LIN {X 0,Y 287.077,Z 619.166,A -85,B 0,C 180,E1 -18390.734,E2 -18390.734} C_VEL
LIN {X 0,Y 290.239,Z 606.893,A -85,B 0,C 180,E1 -18391.78,E2 -18391.78} C_VEL
LIN {X 0,Y 292.756,Z 594.998,A -85,B 0,C 180,E1 -18392.54,E2 -18392.54} C_VEL
LIN {X 0,Y 304.333,Z 525.318,A -85,B 0,C 180,E1 -18395.699,E2 -18395.699} C_VEL
LIN {X 0,Y 304.333,Z 521.564,A -85,B 0,C 180,E1 -18396.179,E2 -18396.179} C_VEL
LIN {X 0,Y 302.945,Z 516.848,A -85,B 0,C 180,E1 -18397.582,E2 -18397.582} C_VEL
LIN {X 0,Y 301.83,Z 513.451,A -85,B 0,C 180,E1 -18398.873,E2 -18398.873} C_VEL
LIN {X 0,Y 300.898,Z 510.648,A -85,B 0,C 180,E1 -18400.235,E2 -18400.235} C_VEL
LIN {X 0,Y 299.797,Z 507.286,A -85,B 0,C 180,E1 -18402.831,E2 -18402.831} C_VEL
LIN {X 0,Y 299.555,Z 506.287,A -85,B 0,C 180,E1 -18404.736,E2 -18404.736} C_VEL
LIN {X 0,Y 300.178,Z 506.371,A -85,B 0,C 180,E1 -18407.424,E2 -18407.424} C_VEL
LIN {X 0,Y 301.713,Z 507.829,A -85,B 0,C 180,E1 -18409.732,E2 -18409.732} C_VEL
LIN {X 0,Y 303.161,Z 509.629,A -85,B 0,C 180,E1 -18411.25,E2 -18411.25} C_VEL
LIN {X 0,Y 303.675,Z 510.855,A -85,B 0,C 180,E1 -18411.798,E2 -18411.798} C_VEL
LIN {X 0,Y 303.632,Z 512.913,A -85,B 0,C 180,E1 -18412.113,E2 -18412.113} C_VEL
LIN {X 0,Y 302.89,Z 524.787,A -85,B 0,C 180,E1 -18413.442,E2 -18413.442} C_VEL
LIN {X 0,Y 301.946,Z 536.286,A -85,B 0,C 180,E1 -18414.495,E2 -18414.495} C_VEL
LIN {X 0,Y 300.792,Z 545.281,A -85,B 0,C 180,E1 -18415.064,E2 -18415.064} C_VEL
LIN {X 0,Y 290.965,Z 604.012,A -85,B 0,C 180,E1 -18417.747,E2 -18417.747} C_VEL
LIN {X 0,Y 287.846,Z 617.704,A -85,B 0,C 180,E1 -18418.592,E2 -18418.592} C_VEL
LIN {X 0,Y 284.125,Z 631.372,A -85,B 0,C 180,E1 -18419.736,E2 -18419.736} C_VEL
LIN {X 0,Y 280.163,Z 643.742,A -85,B 0,C 180,E1 -18421.125,E2 -18421.125} C_VEL
LIN {X 0,Y 276.068,Z 655.019,A -85,B 0,C 180,E1 -18422.727,E2 -18422.727} C_VEL
LIN {X 0,Y 272.401,Z 664.289,A -85,B 0,C 180,E1 -18424.396,E2 -18424.396} C_VEL
LIN {X 0,Y 268.548,Z 673.397,A -85,B 0,C 180,E1 -18426.436,E2 -18426.436} C_VEL
LIN {X 0,Y 265.028,Z 681.094,A -85,B 0,C 180,E1 -18428.616,E2 -18428.616} C_VEL
LIN {X 0,Y 261.491,Z 688.208,A -85,B 0,C 180,E1 -18431.185,E2 -18431.185} C_VEL
LIN {X 0,Y 259.222,Z 692.983,A -85,B 0,C 180,E1 -18433.46,E2 -18433.46} C_VEL
LIN {X 0,Y 257.36,Z 696.664,A -85,B 0,C 180,E1 -18435.772,E2 -18435.772} C_VEL
LIN {X 0,Y 256.3,Z 698.577,A -85,B 0,C 180,E1 -18437.328,E2 -18437.328} C_VEL
LIN {X 0,Y 254.9,Z 701.118,A -85,B 0,C 180,E1 -18440.478,E2 -18440.478} C_VEL
LIN {X 0,Y 254.454,Z 701.775,A -85,B 0,C 180,E1 -18442.062,E2 -18442.062} C_VEL
LIN {X 0,Y 254.086,Z 701.9,A -85,B 0,C 180,E1 -18444.723,E2 -18444.723} C_VEL
LIN {X 0,Y 254.086,Z 701.972,A -85,B 0,C 180,E1 -18446.829,E2 -18446.829} C_VEL
LIN {X 0,Y 254.092,Z 702.588,A -85,B 0,C 180,E1 -18448.415,E2 -18448.415} C_VEL
LIN {X 0,Y 254.1,Z 702.805,A -85,B 0,C 180,E1 -18450,E2 -18450} C_VEL
LIN {X 0,Y 254.061,Z 702.578,A -85,B 0,C 180,E1 -18451.585,E2 -18451.585} C_VEL
LIN {X 0,Y 254.03,Z 701.956,A -85,B 0,C 180,E1 -18453.172,E2 -18453.172} C_VEL
LIN {X 0,Y 254.054,Z 700.586,A -85,B 0,C 180,E1 -18455.199,E2 -18455.199} C_VEL
LIN {X 0,Y 254.338,Z 697.604,A -85,B 0,C 180,E1 -18457.942,E2 -18457.942} C_VEL
LIN {X 0,Y 254.871,Z 693.92,A -85,B 0,C 180,E1 -18460.325,E2 -18460.325} C_VEL
LIN {X 0,Y 255.707,Z 689.104,A -85,B 0,C 180,E1 -18462.702,E2 -18462.702} C_VEL
LIN {X 0,Y 257.053,Z 683.018,A -85,B 0,C 180,E1 -18465.054,E2 -18465.054} C_VEL
LIN {X 0,Y 258.717,Z 675.431,A -85,B 0,C 180,E1 -18467.386,E2 -18467.386} C_VEL
LIN {X 0,Y 260.675,Z 666.14,A -85,B 0,C 180,E1 -18469.695,E2 -18469.695} C_VEL
LIN {X 0,Y 264.028,Z 658.355,A -85,B 0,C 180,E1 -18472.291,E2 -18472.291} C_VEL
LIN {X 0,Y 267.71,Z 650.197,A -85,B 0,C 180,E1 -18474.423,E2 -18474.423} C_VEL
LIN {X 0,Y 271.915,Z 640.356,A -85,B 0,C 180,E1 -18476.478,E2 -18476.478} C_VEL
LIN {X 0,Y 276.223,Z 629.52,A -85,B 0,C 180,E1 -18478.287,E2 -18478.287} C_VEL
LIN {X 0,Y 280.266,Z 618.878,A -85,B 0,C 180,E1 -18479.687,E2 -18479.687} C_VEL
LIN {X 0,Y 284.497,Z 606.061,A -85,B 0,C 180,E1 -18481.043,E2 -18481.043} C_VEL
LIN {X 0,Y 288.605,Z 591.829,A -85,B 0,C 180,E1 -18482.188,E2 -18482.188} C_VEL
LIN {X 0,Y 291.904,Z 578.1,A -85,B 0,C 180,E1 -18483.006,E2 -18483.006} C_VEL
LIN {X 0,Y 295.238,Z 558.089,A -85,B 0,C 180,E1 -18483.963,E2 -18483.963} C_VEL
LIN {X 0,Y 298.029,Z 539.938,A -85,B 0,C 180,E1 -18484.799,E2 -18484.799} C_VEL
LIN {X 0,Y 298.662,Z 531.048,A -85,B 0,C 180,E1 -18485.51,E2 -18485.51} C_VEL
LIN {X 0,Y 299.1,Z 519.805,A -85,B 0,C 180,E1 -18486.643,E2 -18486.643} C_VEL
LIN {X 0,Y 299.142,Z 513.202,A -85,B 0,C 180,E1 -18487.478,E2 -18487.478} C_VEL
LIN {X 0,Y 297.919,Z 508.3,A -85,B 0,C 180,E1 -18488.878,E2 -18488.878} C_VEL
LIN {X 0,Y 296.583,Z 503.001,A -85,B 0,C 180,E1 -18490.821,E2 -18490.821} C_VEL
LIN {X 0,Y 295.391,Z 498.727,A -85,B 0,C 180,E1 -18493.427,E2 -18493.427} C_VEL
LIN {X 0,Y 295.186,Z 496.522,A -85,B 0,C 180,E1 -18495.583,E2 -18495.583} C_VEL
LIN {X 0,Y 295.549,Z 495.761,A -85,B 0,C 180,E1 -18497.491,E2 -18497.491} C_VEL
LIN {X 0,Y 296.945,Z 495.679,A -85,B 0,C 180,E1 -18499.911,E2 -18499.911} C_VEL
LIN {X 0,Y 299.023,Z 498.014,A -85,B 0,C 180,E1 -18502.332,E2 -18502.332} C_VEL
LIN {X 0,Y 301.09,Z 500.788,A -85,B 0,C 180,E1 -18504.056,E2 -18504.056} C_VEL
LIN {X 0,Y 302.889,Z 503.735,A -85,B 0,C 180,E1 -18505.34,E2 -18505.34} C_VEL
LIN {X 0,Y 296.486,Z 542.117,A -85,B 0,C 180,E1 -18507.113,E2 -18507.113} C_VEL
LIN {X 0,Y 294.271,Z 555.53,A -85,B 0,C 180,E1 -18507.9,E2 -18507.9} C_VEL
LIN {X 0,Y 291.464,Z 568.836,A -85,B 0,C 180,E1 -18508.975,E2 -18508.975} C_VEL
LIN {X 0,Y 287.902,Z 582.145,A -85,B 0,C 180,E1 -18510.375,E2 -18510.375} C_VEL
LIN {X 0,Y 284.096,Z 593.977,A -85,B 0,C 180,E1 -18511.964,E2 -18511.964} C_VEL
LIN {X 0,Y 280.51,Z 603.576,A -85,B 0,C 180,E1 -18513.595,E2 -18513.595} C_VEL
LIN {X 0,Y 276.453,Z 613.061,A -85,B 0,C 180,E1 -18515.6,E2 -18515.6} C_VEL
LIN {X 0,Y 272.804,Z 620.742,A -85,B 0,C 180,E1 -18517.667,E2 -18517.667} C_VEL
LIN {X 0,Y 268.959,Z 627.852,A -85,B 0,C 180,E1 -18520.142,E2 -18520.142} C_VEL
LIN {X 0,Y 265.97,Z 632.658,A -85,B 0,C 180,E1 -18522.309,E2 -18522.309} C_VEL
LIN {X 0,Y 263.365,Z 636.317,A -85,B 0,C 180,E1 -18524.523,E2 -18524.523} C_VEL
LIN {X 0,Y 261.81,Z 638.231,A -85,B 0,C 180,E1 -18526.019,E2 -18526.019} C_VEL
LIN {X 0,Y 260.376,Z 639.696,A -85,B 0,C 180,E1 -18527.53,E2 -18527.53} C_VEL
LIN {X 0,Y 259.108,Z 640.706,A -85,B 0,C 180,E1 -18529.055,E2 -18529.055} C_VEL
LIN {X 0,Y 257.274,Z 641.489,A -85,B 0,C 180,E1 -18532.15,E2 -18532.15} C_VEL
LIN {X 0,Y 256.556,Z 641.258,A -85,B 0,C 180,E1 -18533.709,E2 -18533.709} C_VEL
LIN {X 0,Y 255.902,Z 640.608,A -85,B 0,C 180,E1 -18535.274,E2 -18535.274} C_VEL
LIN {X 0,Y 255.396,Z 639.552,A -85,B 0,C 180,E1 -18536.845,E2 -18536.845} C_VEL
LIN {X 0,Y 255.057,Z 638.083,A -85,B 0,C 180,E1 -18538.421,E2 -18538.421} C_VEL
LIN {X 0,Y 254.813,Z 635.042,A -85,B 0,C 180,E1 -18540.79,E2 -18540.79} C_VEL
LIN {X 0,Y 254.821,Z 630.932,A -85,B 0,C 180,E1 -18543.162,E2 -18543.162} C_VEL
LIN {X 0,Y 255.112,Z 625.653,A -85,B 0,C 180,E1 -18545.533,E2 -18545.533} C_VEL
LIN {X 0,Y 255.406,Z 618.206,A -85,B 0,C 180,E1 -18548.177,E2 -18548.177} C_VEL
LIN {X 0,Y 255.836,Z 610.889,A -85,B 0,C 180,E1 -18550.286,E2 -18550.286} C_VEL
LIN {X 0,Y 256.527,Z 602.671,A -85,B 0,C 180,E1 -18552.259,E2 -18552.259} C_VEL
LIN {X 0,Y 257.302,Z 592.708,A -85,B 0,C 180,E1 -18554.231,E2 -18554.231} C_VEL
LIN {X 0,Y 258.225,Z 581.765,A -85,B 0,C 180,E1 -18555.996,E2 -18555.996} C_VEL
LIN {X 0,Y 259.159,Z 569.924,A -85,B 0,C 180,E1 -18557.542,E2 -18557.542} C_VEL
LIN {X 0,Y 259.905,Z 556.354,A -85,B 0,C 180,E1 -18558.935,E2 -18558.935} C_VEL
LIN {X 0,Y 260.686,Z 542.309,A -85,B 0,C 180,E1 -18560.002,E2 -18560.002} C_VEL
LIN {X 0,Y 261.196,Z 527.505,A -85,B 0,C 180,E1 -18560.784,E2 -18560.784} C_VEL
LIN {X 0,Y 263.452,Z 465.935,A -85,B 0,C 180,E1 -18563.408,E2 -18563.408} C_VEL
LIN {X 0,Y 256.196,Z 441.785,A -85,B 0,C 180,E1 -18564.793,E2 -18564.793} C_VEL
LIN {X 0,Y 256.172,Z 441.574,A -85,B 0,C 180,E1 -18565.13,E2 -18565.13} C_VEL
LIN {X 0,Y 256.105,Z 441.585,A -85,B 0,C 180,E1 -18569.601,E2 -18569.601} C_VEL
LIN {X 0,Y 256.07,Z 441.555,A -85,B 0,C 180,E1 -18573.293,E2 -18573.293} C_VEL
LIN {X 0,Y 256.119,Z 441.587,A -85,B 0,C 180,E1 -18577.271,E2 -18577.271} C_VEL
LIN {X 0,Y 256.056,Z 441.571,A -85,B 0,C 180,E1 -18581.203,E2 -18581.203} C_VEL
LIN {X 0,Y 256.046,Z 441.574,A -85,B 0,C 180,E1 -18585.533,E2 -18585.533} C_VEL
LIN {X 0,Y 256.062,Z 441.614,A -85,B 0,C 180,E1 -18589.438,E2 -18589.438} C_VEL
LIN {X 0,Y 259.748,Z 452.744,A -85,B 0,C 180,E1 -18592.964,E2 -18592.964} C_VEL
LIN {X 0,Y 262.936,Z 464.408,A -85,B 0,C 180,E1 -18596.318,E2 -18596.318} C_VEL
LIN {X 0,Y 265.272,Z 474.579,A -85,B 0,C 180,E1 -18599.002,E2 -18599.002} C_VEL
LIN {X 0,Y 268.806,Z 483.491,A -85,B 0,C 180,E1 -18599.734,E2 -18599.734} C_VEL
LIN {X 0,Y 273.159,Z 508.786,A -85,B 0,C 180,E1 -18601.019,E2 -18601.019} C_VEL
LIN {X 0,Y 273.54,Z 513.377,A -85,B 0,C 180,E1 -18601.198,E2 -18601.198} C_VEL
LIN {X 0,Y 271.327,Z 581.026,A -85,B 0,C 180,E1 -18602.941,E2 -18602.941} C_VEL
LIN {X 0,Y 270.624,Z 594.012,A -85,B 0,C 180,E1 -18603.438,E2 -18603.438} C_VEL
LIN {X 0,Y 269.417,Z 606.504,A -85,B 0,C 180,E1 -18604.195,E2 -18604.195} C_VEL
LIN {X 0,Y 268.074,Z 618.207,A -85,B 0,C 180,E1 -18605.199,E2 -18605.199} C_VEL
LIN {X 0,Y 266.286,Z 629.628,A -85,B 0,C 180,E1 -18606.472,E2 -18606.472} C_VEL
LIN {X 0,Y 264.245,Z 641.047,A -85,B 0,C 180,E1 -18608.139,E2 -18608.139} C_VEL
LIN {X 0,Y 262.304,Z 651.222,A -85,B 0,C 180,E1 -18610.025,E2 -18610.025} C_VEL
LIN {X 0,Y 260.486,Z 659.47,A -85,B 0,C 180,E1 -18611.924,E2 -18611.924} C_VEL
LIN {X 0,Y 258.525,Z 667.512,A -85,B 0,C 180,E1 -18614.226,E2 -18614.226} C_VEL
LIN {X 0,Y 257.111,Z 673.973,A -85,B 0,C 180,E1 -18616.565,E2 -18616.565} C_VEL
LIN {X 0,Y 255.91,Z 679.111,A -85,B 0,C 180,E1 -18618.916,E2 -18618.916} C_VEL
LIN {X 0,Y 255.071,Z 683.086,A -85,B 0,C 180,E1 -18621.284,E2 -18621.284} C_VEL
LIN {X 0,Y 254.509,Z 686.142,A -85,B 0,C 180,E1 -18623.777,E2 -18623.777} C_VEL
LIN {X 0,Y 254.163,Z 688.425,A -85,B 0,C 180,E1 -18626.83,E2 -18626.83} C_VEL
LIN {X 0,Y 254.089,Z 689.037,A -85,B 0,C 180,E1 -18628.415,E2 -18628.415} C_VEL
LIN {X 0,Y 254.053,Z 689.27,A -85,B 0,C 180,E1 -18630,E2 -18630} C_VEL
LIN {X 0,Y 254.089,Z 689.073,A -85,B 0,C 180,E1 -18631.585,E2 -18631.585} C_VEL
LIN {X 0,Y 254.163,Z 688.485,A -85,B 0,C 180,E1 -18633.17,E2 -18633.17} C_VEL
LIN {X 0,Y 254.509,Z 686.262,A -85,B 0,C 180,E1 -18636.223,E2 -18636.223} C_VEL
LIN {X 0,Y 255.052,Z 683.266,A -85,B 0,C 180,E1 -18638.717,E2 -18638.717} C_VEL
LIN {X 0,Y 255.854,Z 679.351,A -85,B 0,C 180,E1 -18641.086,E2 -18641.086} C_VEL
LIN {X 0,Y 257.05,Z 674.274,A -85,B 0,C 180,E1 -18643.438,E2 -18643.438} C_VEL
LIN {X 0,Y 258.511,Z 667.873,A -85,B 0,C 180,E1 -18645.775,E2 -18645.775} C_VEL
LIN {X 0,Y 260.448,Z 659.913,A -85,B 0,C 180,E1 -18648.079,E2 -18648.079} C_VEL
LIN {X 0,Y 262.252,Z 651.773,A -85,B 0,C 180,E1 -18649.98,E2 -18649.98} C_VEL
LIN {X 0,Y 264.129,Z 641.749,A -85,B 0,C 180,E1 -18651.871,E2 -18651.871} C_VEL
LIN {X 0,Y 266.247,Z 630.467,A -85,B 0,C 180,E1 -18653.531,E2 -18653.531} C_VEL
LIN {X 0,Y 267.912,Z 619.363,A -85,B 0,C 180,E1 -18654.817,E2 -18654.817} C_VEL
LIN {X 0,Y 269.524,Z 606.769,A -85,B 0,C 180,E1 -18655.898,E2 -18655.898} C_VEL
LIN {X 0,Y 270.653,Z 593.51,A -85,B 0,C 180,E1 -18656.715,E2 -18656.715} C_VEL
LIN {X 0,Y 271.44,Z 580.04,A -85,B 0,C 180,E1 -18657.203,E2 -18657.203} C_VEL
LIN {X 0,Y 273.597,Z 511.499,A -85,B 0,C 180,E1 -18658.977,E2 -18658.977} C_VEL
LIN {X 0,Y 268.862,Z 483.487,A -85,B 0,C 180,E1 -18660.388,E2 -18660.388} C_VEL
LIN {X 0,Y 265.313,Z 474.459,A -85,B 0,C 180,E1 -18661.156,E2 -18661.156} C_VEL
LIN {X 0,Y 262.573,Z 463.006,A -85,B 0,C 180,E1 -18664.2,E2 -18664.2} C_VEL
LIN {X 0,Y 259.4,Z 451.638,A -85,B 0,C 180,E1 -18667.542,E2 -18667.542} C_VEL
LIN {X 0,Y 256.079,Z 441.579,A -85,B 0,C 180,E1 -18670.748,E2 -18670.748} C_VEL
LIN {X 0,Y 256.068,Z 441.58,A -85,B 0,C 180,E1 -18674.472,E2 -18674.472} C_VEL
LIN {X 0,Y 256.057,Z 441.577,A -85,B 0,C 180,E1 -18678.797,E2 -18678.797} C_VEL
LIN {X 0,Y 256.134,Z 441.56,A -85,B 0,C 180,E1 -18682.868,E2 -18682.868} C_VEL
LIN {X 0,Y 256.177,Z 441.704,A -85,B 0,C 180,E1 -18686.504,E2 -18686.504} C_VEL
LIN {X 0,Y 259.476,Z 457.293,A -85,B 0,C 180,E1 -18690.427,E2 -18690.427} C_VEL
LIN {X 0,Y 259.871,Z 459.167,A -85,B 0,C 180,E1 -18690.894,E2 -18690.894} C_VEL
LIN {X 0,Y 259.705,Z 461.871,A -85,B 0,C 180,E1 -18691.517,E2 -18691.517} C_VEL
LIN {X 0,Y 257.424,Z 466.463,A -85,B 0,C 180,E1 -18692.459,E2 -18692.459} C_VEL
LIN {X 0,Y 254.283,Z 472.076,A -85,B 0,C 180,E1 -18693.606,E2 -18693.606} C_VEL
LIN {X 0,Y 253.836,Z 473.979,A -85,B 0,C 180,E1 -18694.031,E2 -18694.031} C_VEL
LIN {X 0,Y 253.691,Z 475.369,A -85,B 0,C 180,E1 -18694.351,E2 -18694.351} C_VEL
LIN {X 0,Y 255.615,Z 497.34,A -85,B 0,C 180,E1 -18695.456,E2 -18695.456} C_VEL
LIN {X 0,Y 256.793,Z 508.953,A -85,B 0,C 180,E1 -18696.03,E2 -18696.03} C_VEL
LIN {X 0,Y 253.537,Z 588.135,A -85,B 0,C 180,E1 -18699.568,E2 -18699.568} C_VEL
LIN {X 0,Y 252.757,Z 601.971,A -85,B 0,C 180,E1 -18700.509,E2 -18700.509} C_VEL
LIN {X 0,Y 251.763,Z 616.05,A -85,B 0,C 180,E1 -18701.835,E2 -18701.835} C_VEL
LIN {X 0,Y 250.796,Z 628.063,A -85,B 0,C 180,E1 -18703.307,E2 -18703.307} C_VEL
LIN {X 0,Y 249.942,Z 638.62,A -85,B 0,C 180,E1 -18704.924,E2 -18704.924} C_VEL
LIN {X 0,Y 249.003,Z 649.403,A -85,B 0,C 180,E1 -18706.95,E2 -18706.95} C_VEL
LIN {X 0,Y 248.261,Z 658.232,A -85,B 0,C 180,E1 -18708.984,E2 -18708.984} C_VEL
LIN {X 0,Y 247.74,Z 665.596,A -85,B 0,C 180,E1 -18711.024,E2 -18711.024} C_VEL
LIN {X 0,Y 247.263,Z 672.819,A -85,B 0,C 180,E1 -18713.472,E2 -18713.472} C_VEL
LIN {X 0,Y 247.076,Z 678.574,A -85,B 0,C 180,E1 -18715.922,E2 -18715.922} C_VEL
LIN {X 0,Y 247.004,Z 683.043,A -85,B 0,C 180,E1 -18718.369,E2 -18718.369} C_VEL
LIN {X 0,Y 246.976,Z 685.387,A -85,B 0,C 180,E1 -18720,E2 -18720} C_VEL
LIN {X 0,Y 247.039,Z 687.225,A -85,B 0,C 180,E1 -18721.63,E2 -18721.63} C_VEL
LIN {X 0,Y 247.113,Z 688.639,A -85,B 0,C 180,E1 -18723.261,E2 -18723.261} C_VEL
LIN {X 0,Y 247.328,Z 689.651,A -85,B 0,C 180,E1 -18724.89,E2 -18724.89} C_VEL
LIN {X 0,Y 247.853,Z 690.298,A -85,B 0,C 180,E1 -18727.047,E2 -18727.047} C_VEL
LIN {X 0,Y 248.877,Z 690.108,A -85,B 0,C 180,E1 -18729.755,E2 -18729.755} C_VEL
LIN {X 0,Y 249.738,Z 689.451,A -85,B 0,C 180,E1 -18731.361,E2 -18731.361} C_VEL
LIN {X 0,Y 252,Z 686.855,A -85,B 0,C 180,E1 -18734.537,E2 -18734.537} C_VEL
LIN {X 0,Y 254.163,Z 683.832,A -85,B 0,C 180,E1 -18736.878,E2 -18736.878} C_VEL
LIN {X 0,Y 256.926,Z 679.724,A -85,B 0,C 180,E1 -18739.163,E2 -18739.163} C_VEL
LIN {X 0,Y 260.542,Z 673.584,A -85,B 0,C 180,E1 -18741.771,E2 -18741.771} C_VEL
LIN {X 0,Y 264.87,Z 665.645,A -85,B 0,C 180,E1 -18744.285,E2 -18744.285} C_VEL
LIN {X 0,Y 269.718,Z 655.632,A -85,B 0,C 180,E1 -18746.71,E2 -18746.71} C_VEL
LIN {X 0,Y 273.936,Z 645.888,A -85,B 0,C 180,E1 -18748.544,E2 -18748.544} C_VEL
LIN {X 0,Y 278.06,Z 635.222,A -85,B 0,C 180,E1 -18750.155,E2 -18750.155} C_VEL
LIN {X 0,Y 282.027,Z 623.444,A -85,B 0,C 180,E1 -18751.555,E2 -18751.555} C_VEL
LIN {X 0,Y 285.76,Z 610.37,A -85,B 0,C 180,E1 -18752.757,E2 -18752.757} C_VEL
LIN {X 0,Y 288.729,Z 597.939,A -85,B 0,C 180,E1 -18753.625,E2 -18753.625} C_VEL
LIN {X 0,Y 292.053,Z 579.862,A -85,B 0,C 180,E1 -18754.509,E2 -18754.509} C_VEL
LIN {X 0,Y 301.327,Z 527.843,A -85,B 0,C 180,E1 -18756.832,E2 -18756.832} C_VEL
LIN {X 0,Y 301.333,Z 526.347,A -85,B 0,C 180,E1 -18757.043,E2 -18757.043} C_VEL
LIN {X 0,Y 300.052,Z 521.266,A -85,B 0,C 180,E1 -18758.659,E2 -18758.659} C_VEL
LIN {X 0,Y 298.862,Z 517.239,A -85,B 0,C 180,E1 -18760.539,E2 -18760.539} C_VEL
LIN {X 0,Y 297.985,Z 514.079,A -85,B 0,C 180,E1 -18763.018,E2 -18763.018} C_VEL
LIN {X 0,Y 297.834,Z 513.058,A -85,B 0,C 180,E1 -18765.065,E2 -18765.065} C_VEL
LIN {X 0,Y 298.615,Z 513.366,A -85,B 0,C 180,E1 -18767.752,E2 -18767.752} C_VEL
LIN {X 0,Y 300.482,Z 515.35,A -85,B 0,C 180,E1 -18770.352,E2 -18770.352} C_VEL
LIN {X 0,Y 301.093,Z 516.394,A -85,B 0,C 180,E1 -18771.039,E2 -18771.039} C_VEL
LIN {X 0,Y 300.071,Z 527.53,A -85,B 0,C 180,E1 -18772.322,E2 -18772.322} C_VEL
LIN {X 0,Y 298.904,Z 538.933,A -85,B 0,C 180,E1 -18773.371,E2 -18773.371} C_VEL
LIN {X 0,Y 297.828,Z 546.265,A -85,B 0,C 180,E1 -18773.847,E2 -18773.847} C_VEL
LIN {X 0,Y 287.713,Z 602.83,A -85,B 0,C 180,E1 -18776.459,E2 -18776.459} C_VEL
LIN {X 0,Y 284.334,Z 617.057,A -85,B 0,C 180,E1 -18777.316,E2 -18777.316} C_VEL
LIN {X 0,Y 280.446,Z 630.316,A -85,B 0,C 180,E1 -18778.417,E2 -18778.417} C_VEL
LIN {X 0,Y 276.555,Z 641.731,A -85,B 0,C 180,E1 -18779.663,E2 -18779.663} C_VEL
LIN {X 0,Y 272.14,Z 653.254,A -85,B 0,C 180,E1 -18781.25,E2 -18781.25} C_VEL
LIN {X 0,Y 267.744,Z 663.508,A -85,B 0,C 180,E1 -18783.077,E2 -18783.077} C_VEL
LIN {X 0,Y 263.233,Z 673.376,A -85,B 0,C 180,E1 -18785.3,E2 -18785.3} C_VEL
LIN {X 0,Y 259.125,Z 681.503,A -85,B 0,C 180,E1 -18787.684,E2 -18787.684} C_VEL
LIN {X 0,Y 255.927,Z 687.543,A -85,B 0,C 180,E1 -18789.924,E2 -18789.924} C_VEL
LIN {X 0,Y 253.131,Z 692.371,A -85,B 0,C 180,E1 -18792.217,E2 -18792.217} C_VEL
LIN {X 0,Y 251.088,Z 696.131,A -85,B 0,C 180,E1 -18794.579,E2 -18794.579} C_VEL
LIN {X 0,Y 249.392,Z 698.893,A -85,B 0,C 180,E1 -18796.971,E2 -18796.971} C_VEL
LIN {X 0,Y 248.536,Z 700.231,A -85,B 0,C 180,E1 -18798.583,E2 -18798.583} C_VEL
LIN {X 0,Y 247.886,Z 701.13,A -85,B 0,C 180,E1 -18800.206,E2 -18800.206} C_VEL
LIN {X 0,Y 247.113,Z 701.707,A -85,B 0,C 180,E1 -18803.468,E2 -18803.468} C_VEL
LIN {X 0,Y 246.982,Z 701.294,A -85,B 0,C 180,E1 -18805.845,E2 -18805.845} C_VEL
LIN {X 0,Y 247,Z 702.399,A -85,B 0,C 180,E1 -18808.37,E2 -18808.37} C_VEL
LIN {X 0,Y 247.027,Z 702.617,A -85,B 0,C 180,E1 -18810,E2 -18810} C_VEL
LIN {X 0,Y 246.968,Z 702.388,A -85,B 0,C 180,E1 -18811.631,E2 -18811.631} C_VEL
LIN {X 0,Y 246.928,Z 701.766,A -85,B 0,C 180,E1 -18813.263,E2 -18813.263} C_VEL
LIN {X 0,Y 246.951,Z 700.622,A -85,B 0,C 180,E1 -18815.082,E2 -18815.082} C_VEL
LIN {X 0,Y 247.285,Z 697.414,A -85,B 0,C 180,E1 -18818.17,E2 -18818.17} C_VEL
LIN {X 0,Y 247.852,Z 693.73,A -85,B 0,C 180,E1 -18820.621,E2 -18820.621} C_VEL
LIN {X 0,Y 248.74,Z 688.914,A -85,B 0,C 180,E1 -18823.064,E2 -18823.064} C_VEL
LIN {X 0,Y 250.185,Z 682.83,A -85,B 0,C 180,E1 -18825.478,E2 -18825.478} C_VEL
LIN {X 0,Y 251.947,Z 675.243,A -85,B 0,C 180,E1 -18827.869,E2 -18827.869} C_VEL
LIN {X 0,Y 253.619,Z 667.577,A -85,B 0,C 180,E1 -18829.844,E2 -18829.844} C_VEL
LIN {X 0,Y 257.026,Z 660.451,A -85,B 0,C 180,E1 -18832.508,E2 -18832.508} C_VEL
LIN {X 0,Y 260.696,Z 652.975,A -85,B 0,C 180,E1 -18834.7,E2 -18834.7} C_VEL
LIN {X 0,Y 264.966,Z 643.993,A -85,B 0,C 180,E1 -18836.802,E2 -18836.802} C_VEL
LIN {X 0,Y 269.758,Z 633.166,A -85,B 0,C 180,E1 -18838.815,E2 -18838.815} C_VEL
LIN {X 0,Y 274.279,Z 622.331,A -85,B 0,C 180,E1 -18840.402,E2 -18840.402} C_VEL
LIN {X 0,Y 279.187,Z 609.141,A -85,B 0,C 180,E1 -18841.913,E2 -18841.913} C_VEL
LIN {X 0,Y 283.967,Z 594.285,A -85,B 0,C 180,E1 -18843.201,E2 -18843.201} C_VEL
LIN {X 0,Y 287.963,Z 579.312,A -85,B 0,C 180,E1 -18844.148,E2 -18844.148} C_VEL
LIN {X 0,Y 291.002,Z 563.528,A -85,B 0,C 180,E1 -18844.948,E2 -18844.948} C_VEL
LIN {X 0,Y 294.632,Z 541.553,A -85,B 0,C 180,E1 -18845.967,E2 -18845.967} C_VEL
LIN {X 0,Y 295.381,Z 533.329,A -85,B 0,C 180,E1 -18846.643,E2 -18846.643} C_VEL
LIN {X 0,Y 296.032,Z 522.993,A -85,B 0,C 180,E1 -18847.709,E2 -18847.709} C_VEL
LIN {X 0,Y 296.169,Z 517.912,A -85,B 0,C 180,E1 -18848.381,E2 -18848.381} C_VEL
LIN {X 0,Y 295.398,Z 514.197,A -85,B 0,C 180,E1 -18849.472,E2 -18849.472} C_VEL
LIN {X 0,Y 294.374,Z 509.333,A -85,B 0,C 180,E1 -18851.283,E2 -18851.283} C_VEL
LIN {X 0,Y 293.436,Z 505.161,A -85,B 0,C 180,E1 -18853.88,E2 -18853.88} C_VEL
LIN {X 0,Y 293.406,Z 503.183,A -85,B 0,C 180,E1 -18856.001,E2 -18856.001} C_VEL
LIN {X 0,Y 293.926,Z 502.574,A -85,B 0,C 180,E1 -18857.971,E2 -18857.971} C_VEL
LIN {X 0,Y 295.17,Z 502.637,A -85,B 0,C 180,E1 -18859.994,E2 -18859.994} C_VEL
LIN {X 0,Y 297.024,Z 504.819,A -85,B 0,C 180,E1 -18862.199,E2 -18862.199} C_VEL
LIN {X 0,Y 298.702,Z 507.233,A -85,B 0,C 180,E1 -18863.694,E2 -18863.694} C_VEL
LIN {X 0,Y 299.454,Z 508.375,A -85,B 0,C 180,E1 -18864.284,E2 -18864.284} C_VEL
LIN {X 0,Y 293.342,Z 542.603,A -85,B 0,C 180,E1 -18865.878,E2 -18865.878} C_VEL
LIN {X 0,Y 290.941,Z 556.061,A -85,B 0,C 180,E1 -18866.664,E2 -18866.664} C_VEL
LIN {X 0,Y 287.939,Z 569.29,A -85,B 0,C 180,E1 -18867.729,E2 -18867.729} C_VEL
LIN {X 0,Y 284.155,Z 582.557,A -85,B 0,C 180,E1 -18869.122,E2 -18869.122} C_VEL
LIN {X 0,Y 280.058,Z 594.365,A -85,B 0,C 180,E1 -18870.702,E2 -18870.702} C_VEL
LIN {X 0,Y 275.494,Z 605.766,A -85,B 0,C 180,E1 -18872.665,E2 -18872.665} C_VEL
LIN {X 0,Y 271.198,Z 614.938,A -85,B 0,C 180,E1 -18874.685,E2 -18874.685} C_VEL
LIN {X 0,Y 266.679,Z 623.488,A -85,B 0,C 180,E1 -18877.125,E2 -18877.125} C_VEL
LIN {X 0,Y 262.644,Z 630.191,A -85,B 0,C 180,E1 -18879.643,E2 -18879.643} C_VEL
LIN {X 0,Y 258.53,Z 635.891,A -85,B 0,C 180,E1 -18882.601,E2 -18882.601} C_VEL
LIN {X 0,Y 256.737,Z 638.066,A -85,B 0,C 180,E1 -18884.113,E2 -18884.113} C_VEL
LIN {X 0,Y 255.085,Z 639.749,A -85,B 0,C 180,E1 -18885.643,E2 -18885.643} C_VEL
LIN {X 0,Y 252.245,Z 641.902,A -85,B 0,C 180,E1 -18888.753,E2 -18888.753} C_VEL
LIN {X 0,Y 251.184,Z 642.346,A -85,B 0,C 180,E1 -18890.336,E2 -18890.336} C_VEL
LIN {X 0,Y 250.32,Z 642.351,A -85,B 0,C 180,E1 -18891.93,E2 -18891.93} C_VEL
LIN {X 0,Y 248.866,Z 641.195,A -85,B 0,C 180,E1 -18895.14,E2 -18895.14} C_VEL
LIN {X 0,Y 248.347,Z 639.989,A -85,B 0,C 180,E1 -18896.755,E2 -18896.755} C_VEL
LIN {X 0,Y 247.84,Z 637.374,A -85,B 0,C 180,E1 -18899.188,E2 -18899.188} C_VEL
LIN {X 0,Y 247.677,Z 633.752,A -85,B 0,C 180,E1 -18901.626,E2 -18901.626} C_VEL
LIN {X 0,Y 247.842,Z 629.041,A -85,B 0,C 180,E1 -18904.065,E2 -18904.065} C_VEL
LIN {X 0,Y 248.042,Z 623.076,A -85,B 0,C 180,E1 -18906.508,E2 -18906.508} C_VEL
LIN {X 0,Y 248.474,Z 615.662,A -85,B 0,C 180,E1 -18908.95,E2 -18908.95} C_VEL
LIN {X 0,Y 249.114,Z 606.528,A -85,B 0,C 180,E1 -18911.39,E2 -18911.39} C_VEL
LIN {X 0,Y 249.938,Z 596.193,A -85,B 0,C 180,E1 -18913.621,E2 -18913.621} C_VEL
LIN {X 0,Y 250.933,Z 584.644,A -85,B 0,C 180,E1 -18915.639,E2 -18915.639} C_VEL
LIN {X 0,Y 251.926,Z 571.664,A -85,B 0,C 180,E1 -18917.451,E2 -18917.451} C_VEL
LIN {X 0,Y 252.767,Z 558.638,A -85,B 0,C 180,E1 -18918.866,E2 -18918.866} C_VEL
LIN {X 0,Y 253.448,Z 545.454,A -85,B 0,C 180,E1 -18919.964,E2 -18919.964} C_VEL
LIN {X 0,Y 254.013,Z 531.825,A -85,B 0,C 180,E1 -18920.763,E2 -18920.763} C_VEL
LIN {X 0,Y 256.426,Z 467.128,A -85,B 0,C 180,E1 -18923.626,E2 -18923.626} C_VEL
LIN {X 0,Y 249.36,Z 443.589,A -85,B 0,C 180,E1 -18925.029,E2 -18925.029} C_VEL
LIN {X 0,Y 249.134,Z 442.451,A -85,B 0,C 180,E1 -18925.118,E2 -18925.118} C_VEL
LIN {X 0,Y 249.075,Z 442.455,A -85,B 0,C 180,E1 -18928.989,E2 -18928.989} C_VEL
LIN {X 0,Y 249.032,Z 442.437,A -85,B 0,C 180,E1 -18932.426,E2 -18932.426} C_VEL
LIN {X 0,Y 249.051,Z 442.459,A -85,B 0,C 180,E1 -18936.342,E2 -18936.342} C_VEL
LIN {X 0,Y 249.008,Z 442.445,A -85,B 0,C 180,E1 -18940.478,E2 -18940.478} C_VEL
LIN {X 0,Y 248.997,Z 442.456,A -85,B 0,C 180,E1 -18944.881,E2 -18944.881} C_VEL
LIN {X 0,Y 249.028,Z 442.556,A -85,B 0,C 180,E1 -18948.371,E2 -18948.371} C_VEL
LIN {X 0,Y 253.112,Z 454.697,A -85,B 0,C 180,E1 -18952.348,E2 -18952.348} C_VEL
LIN {X 0,Y 255.99,Z 465.115,A -85,B 0,C 180,E1 -18955.45,E2 -18955.45} C_VEL
LIN {X 0,Y 258.437,Z 475.052,A -85,B 0,C 180,E1 -18958.107,E2 -18958.107} C_VEL
LIN {X 0,Y 262.97,Z 486.165,A -85,B 0,C 180,E1 -18959.071,E2 -18959.071} C_VEL
LIN {X 0,Y 267.116,Z 510.952,A -85,B 0,C 180,E1 -18960.361,E2 -18960.361} C_VEL
LIN {X 0,Y 267.321,Z 514.414,A -85,B 0,C 180,E1 -18960.492,E2 -18960.492} C_VEL
LIN {X 0,Y 264.904,Z 584.093,A -85,B 0,C 180,E1 -18962.336,E2 -18962.336} C_VEL
LIN {X 0,Y 263.991,Z 597.546,A -85,B 0,C 180,E1 -18962.93,E2 -18962.93} C_VEL
LIN {X 0,Y 262.785,Z 609.129,A -85,B 0,C 180,E1 -18963.707,E2 -18963.707} C_VEL
LIN {X 0,Y 261.338,Z 620.228,A -85,B 0,C 180,E1 -18964.728,E2 -18964.728} C_VEL
LIN {X 0,Y 259.537,Z 631.188,A -85,B 0,C 180,E1 -18966.034,E2 -18966.034} C_VEL
LIN {X 0,Y 257.429,Z 642.482,A -85,B 0,C 180,E1 -18967.762,E2 -18967.762} C_VEL
LIN {X 0,Y 255.628,Z 651.408,A -85,B 0,C 180,E1 -18969.48,E2 -18969.48} C_VEL
LIN {X 0,Y 253.754,Z 659.657,A -85,B 0,C 180,E1 -18971.427,E2 -18971.427} C_VEL
LIN {X 0,Y 251.7,Z 667.7,A -85,B 0,C 180,E1 -18973.786,E2 -18973.786} C_VEL
LIN {X 0,Y 250.196,Z 674.162,A -85,B 0,C 180,E1 -18976.186,E2 -18976.186} C_VEL
LIN {X 0,Y 248.928,Z 679.301,A -85,B 0,C 180,E1 -18978.601,E2 -18978.601} C_VEL
LIN {X 0,Y 248.061,Z 683.275,A -85,B 0,C 180,E1 -18981.035,E2 -18981.035} C_VEL
LIN {X 0,Y 247.388,Z 686.597,A -85,B 0,C 180,E1 -18983.887,E2 -18983.887} C_VEL
LIN {X 0,Y 247.084,Z 688.614,A -85,B 0,C 180,E1 -18986.739,E2 -18986.739} C_VEL
LIN {X 0,Y 247,Z 689.226,A -85,B 0,C 180,E1 -18988.37,E2 -18988.37} C_VEL
LIN {X 0,Y 246.983,Z 689.458,A -85,B 0,C 180,E1 -18990,E2 -18990} C_VEL
LIN {X 0,Y 246.999,Z 689.262,A -85,B 0,C 180,E1 -18991.63,E2 -18991.63} C_VEL
LIN {X 0,Y 247.084,Z 688.674,A -85,B 0,C 180,E1 -18993.261,E2 -18993.261} C_VEL
LIN {X 0,Y 247.418,Z 686.646,A -85,B 0,C 180,E1 -18996.178,E2 -18996.178} C_VEL
LIN {X 0,Y 248.043,Z 683.453,A -85,B 0,C 180,E1 -18998.965,E2 -18998.965} C_VEL
LIN {X 0,Y 248.882,Z 679.538,A -85,B 0,C 180,E1 -19001.401,E2 -19001.401} C_VEL
LIN {X 0,Y 250.143,Z 674.459,A -85,B 0,C 180,E1 -19003.817,E2 -19003.817} C_VEL
LIN {X 0,Y 251.687,Z 668.057,A -85,B 0,C 180,E1 -19006.215,E2 -19006.215} C_VEL
LIN {X 0,Y 253.713,Z 660.095,A -85,B 0,C 180,E1 -19008.576,E2 -19008.576} C_VEL
LIN {X 0,Y 255.684,Z 651.422,A -85,B 0,C 180,E1 -19010.641,E2 -19010.641} C_VEL
LIN {X 0,Y 257.781,Z 640.785,A -85,B 0,C 180,E1 -19012.65,E2 -19012.65} C_VEL
LIN {X 0,Y 259.744,Z 630.639,A -85,B 0,C 180,E1 -19014.157,E2 -19014.157} C_VEL
LIN {X 0,Y 261.502,Z 619.525,A -85,B 0,C 180,E1 -19015.468,E2 -19015.468} C_VEL
LIN {X 0,Y 263.172,Z 606.92,A -85,B 0,C 180,E1 -19016.571,E2 -19016.571} C_VEL
LIN {X 0,Y 264.28,Z 594.505,A -85,B 0,C 180,E1 -19017.359,E2 -19017.359} C_VEL
LIN {X 0,Y 265.089,Z 581.756,A -85,B 0,C 180,E1 -19017.858,E2 -19017.858} C_VEL
LIN {X 0,Y 267.356,Z 512.299,A -85,B 0,C 180,E1 -19019.697,E2 -19019.697} C_VEL
LIN {X 0,Y 263.024,Z 486.291,A -85,B 0,C 180,E1 -19021.05,E2 -19021.05} C_VEL
LIN {X 0,Y 259.387,Z 477.193,A -85,B 0,C 180,E1 -19021.827,E2 -19021.827} C_VEL
LIN {X 0,Y 258.343,Z 474.654,A -85,B 0,C 180,E1 -19022.088,E2 -19022.088} C_VEL
LIN {X 0,Y 255.223,Z 462.068,A -85,B 0,C 180,E1 -19025.571,E2 -19025.571} C_VEL
LIN {X 0,Y 252.191,Z 451.844,A -85,B 0,C 180,E1 -19028.712,E2 -19028.712} C_VEL
LIN {X 0,Y 249.047,Z 442.465,A -85,B 0,C 180,E1 -19031.813,E2 -19031.813} C_VEL
LIN {X 0,Y 249.012,Z 442.465,A -85,B 0,C 180,E1 -19035.122,E2 -19035.122} C_VEL
LIN {X 0,Y 249.008,Z 442.461,A -85,B 0,C 180,E1 -19039.522,E2 -19039.522} C_VEL
LIN {X 0,Y 249.06,Z 442.439,A -85,B 0,C 180,E1 -19043.659,E2 -19043.659} C_VEL
LIN {X 0,Y 249.105,Z 442.525,A -85,B 0,C 180,E1 -19046.189,E2 -19046.189} C_VEL
LIN {X 0,Y 252.601,Z 458.976,A -85,B 0,C 180,E1 -19050.406,E2 -19050.406} C_VEL
LIN {X 0,Y 254.264,Z 467.393,A -85,B 0,C 180,E1 -19052.499,E2 -19052.499} C_VEL
LIN {X 0,Y 253.836,Z 473.979,A -85,B 0,C 180,E1 -19054.031,E2 -19054.031} C_VEL
LIN {X 0,Y 253.059,Z 476.27,A -85,B 0,C 180,E1 -19054.338,E2 -19054.338} C_VEL
LIN {X 0,Y 248.374,Z 485.16,A -85,B 0,C 180,E1 -19054.587,E2 -19054.587} C_VEL
LIN {X 0,Y 247.287,Z 489.146,A -85,B 0,C 180,E1 -19054.708,E2 -19054.708} C_VEL
LIN {X 0,Y 247.382,Z 494.266,A -85,B 0,C 180,E1 -19054.926,E2 -19054.926} C_VEL
LIN {X 0,Y 249.378,Z 504.404,A -85,B 0,C 180,E1 -19055.535,E2 -19055.535} C_VEL
LIN {X 0,Y 249.79,Z 509.87,A -85,B 0,C 180,E1 -19055.805,E2 -19055.805} C_VEL
LIN {X 0,Y 246.467,Z 587.25,A -85,B 0,C 180,E1 -19059.391,E2 -19059.391} C_VEL
LIN {X 0,Y 245.663,Z 602.164,A -85,B 0,C 180,E1 -19060.437,E2 -19060.437} C_VEL
LIN {X 0,Y 244.664,Z 616.073,A -85,B 0,C 180,E1 -19061.797,E2 -19061.797} C_VEL
LIN {X 0,Y 243.733,Z 627.57,A -85,B 0,C 180,E1 -19063.241,E2 -19063.241} C_VEL
LIN {X 0,Y 242.949,Z 637.017,A -85,B 0,C 180,E1 -19064.694,E2 -19064.694} C_VEL
LIN {X 0,Y 242.074,Z 647.129,A -85,B 0,C 180,E1 -19066.57,E2 -19066.57} C_VEL
LIN {X 0,Y 241.316,Z 656.446,A -85,B 0,C 180,E1 -19068.663,E2 -19068.663} C_VEL
LIN {X 0,Y 240.642,Z 665.498,A -85,B 0,C 180,E1 -19071.18,E2 -19071.18} C_VEL
LIN {X 0,Y 240.24,Z 671.67,A -85,B 0,C 180,E1 -19073.28,E2 -19073.28} C_VEL
LIN {X 0,Y 240.005,Z 677.695,A -85,B 0,C 180,E1 -19075.802,E2 -19075.802} C_VEL
LIN {X 0,Y 239.941,Z 682.398,A -85,B 0,C 180,E1 -19078.321,E2 -19078.321} C_VEL
LIN {X 0,Y 239.915,Z 685.946,A -85,B 0,C 180,E1 -19080.839,E2 -19080.839} C_VEL
LIN {X 0,Y 240.039,Z 688.465,A -85,B 0,C 180,E1 -19083.357,E2 -19083.357} C_VEL
LIN {X 0,Y 240.648,Z 690.307,A -85,B 0,C 180,E1 -19086.708,E2 -19086.708} C_VEL
LIN {X 0,Y 241.205,Z 690.629,A -85,B 0,C 180,E1 -19088.377,E2 -19088.377} C_VEL
LIN {X 0,Y 242.804,Z 689.994,A -85,B 0,C 180,E1 -19091.69,E2 -19091.69} C_VEL
LIN {X 0,Y 243.932,Z 689.102,A -85,B 0,C 180,E1 -19093.326,E2 -19093.326} C_VEL
LIN {X 0,Y 245.207,Z 687.785,A -85,B 0,C 180,E1 -19094.949,E2 -19094.949} C_VEL
LIN {X 0,Y 247.481,Z 685.016,A -85,B 0,C 180,E1 -19097.348,E2 -19097.348} C_VEL
LIN {X 0,Y 251.435,Z 679.754,A -85,B 0,C 180,E1 -19100.45,E2 -19100.45} C_VEL
LIN {X 0,Y 254.824,Z 674.531,A -85,B 0,C 180,E1 -19102.713,E2 -19102.713} C_VEL
LIN {X 0,Y 259.405,Z 666.844,A -85,B 0,C 180,E1 -19105.259,E2 -19105.259} C_VEL
LIN {X 0,Y 263.8,Z 658.663,A -85,B 0,C 180,E1 -19107.359,E2 -19107.359} C_VEL
LIN {X 0,Y 268.584,Z 648.709,A -85,B 0,C 180,E1 -19109.382,E2 -19109.382} C_VEL
LIN {X 0,Y 272.876,Z 638.639,A -85,B 0,C 180,E1 -19111.005,E2 -19111.005} C_VEL
LIN {X 0,Y 277.518,Z 626.351,A -85,B 0,C 180,E1 -19112.557,E2 -19112.557} C_VEL
LIN {X 0,Y 281.406,Z 614.107,A -85,B 0,C 180,E1 -19113.758,E2 -19113.758} C_VEL
LIN {X 0,Y 285.024,Z 600.428,A -85,B 0,C 180,E1 -19114.765,E2 -19114.765} C_VEL
LIN {X 0,Y 288.229,Z 585.259,A -85,B 0,C 180,E1 -19115.549,E2 -19115.549} C_VEL
LIN {X 0,Y 298.518,Z 530.949,A -85,B 0,C 180,E1 -19117.999,E2 -19117.999} C_VEL
LIN {X 0,Y 297.555,Z 526.692,A -85,B 0,C 180,E1 -19119.498,E2 -19119.498} C_VEL
LIN {X 0,Y 296.848,Z 523.834,A -85,B 0,C 180,E1 -19120.865,E2 -19120.865} C_VEL
LIN {X 0,Y 296.147,Z 520.971,A -85,B 0,C 180,E1 -19123.103,E2 -19123.103} C_VEL
LIN {X 0,Y 296.023,Z 520.085,A -85,B 0,C 180,E1 -19124.582,E2 -19124.582} C_VEL
LIN {X 0,Y 296.565,Z 520.07,A -85,B 0,C 180,E1 -19127.277,E2 -19127.277} C_VEL
LIN {X 0,Y 297.9,Z 521.435,A -85,B 0,C 180,E1 -19129.474,E2 -19129.474} C_VEL
LIN {X 0,Y 298.535,Z 522.312,A -85,B 0,C 180,E1 -19130.261,E2 -19130.261} C_VEL
LIN {X 0,Y 297.116,Z 534.156,A -85,B 0,C 180,E1 -19131.559,E2 -19131.559} C_VEL
LIN {X 0,Y 296.051,Z 541.903,A -85,B 0,C 180,E1 -19132.232,E2 -19132.232} C_VEL
LIN {X 0,Y 294.955,Z 548.351,A -85,B 0,C 180,E1 -19132.646,E2 -19132.646} C_VEL
LIN {X 0,Y 284.27,Z 604.118,A -85,B 0,C 180,E1 -19135.237,E2 -19135.237} C_VEL
LIN {X 0,Y 280.972,Z 616.964,A -85,B 0,C 180,E1 -19136.026,E2 -19136.026} C_VEL
LIN {X 0,Y 277.452,Z 628.204,A -85,B 0,C 180,E1 -19136.942,E2 -19136.942} C_VEL
LIN {X 0,Y 273.255,Z 640.047,A -85,B 0,C 180,E1 -19138.18,E2 -19138.18} C_VEL
LIN {X 0,Y 268.809,Z 650.987,A -85,B 0,C 180,E1 -19139.65,E2 -19139.65} C_VEL
LIN {X 0,Y 264.146,Z 661.271,A -85,B 0,C 180,E1 -19141.385,E2 -19141.385} C_VEL
LIN {X 0,Y 259.476,Z 670.786,A -85,B 0,C 180,E1 -19143.454,E2 -19143.454} C_VEL
LIN {X 0,Y 254.646,Z 679.84,A -85,B 0,C 180,E1 -19145.986,E2 -19145.986} C_VEL
LIN {X 0,Y 250.362,Z 686.975,A -85,B 0,C 180,E1 -19148.597,E2 -19148.597} C_VEL
LIN {X 0,Y 247.402,Z 691.839,A -85,B 0,C 180,E1 -19150.932,E2 -19150.932} C_VEL
LIN {X 0,Y 244.918,Z 695.635,A -85,B 0,C 180,E1 -19153.324,E2 -19153.324} C_VEL
LIN {X 0,Y 243.62,Z 697.627,A -85,B 0,C 180,E1 -19154.952,E2 -19154.952} C_VEL
LIN {X 0,Y 242.477,Z 699.192,A -85,B 0,C 180,E1 -19156.593,E2 -19156.593} C_VEL
LIN {X 0,Y 240.89,Z 701.092,A -85,B 0,C 180,E1 -19159.918,E2 -19159.918} C_VEL
LIN {X 0,Y 240.383,Z 701.457,A -85,B 0,C 180,E1 -19161.594,E2 -19161.594} C_VEL
LIN {X 0,Y 239.952,Z 700.959,A -85,B 0,C 180,E1 -19164.77,E2 -19164.77} C_VEL
LIN {X 0,Y 239.911,Z 700.8,A -85,B 0,C 180,E1 -19165.274,E2 -19165.274} C_VEL
LIN {X 0,Y 239.909,Z 702.21,A -85,B 0,C 180,E1 -19168.321,E2 -19168.321} C_VEL
LIN {X 0,Y 239.956,Z 702.428,A -85,B 0,C 180,E1 -19170,E2 -19170} C_VEL
LIN {X 0,Y 239.877,Z 702.199,A -85,B 0,C 180,E1 -19171.679,E2 -19171.679} C_VEL
LIN {X 0,Y 239.844,Z 700.631,A -85,B 0,C 180,E1 -19174.94,E2 -19174.94} C_VEL
LIN {X 0,Y 239.99,Z 699.123,A -85,B 0,C 180,E1 -19176.727,E2 -19176.727} C_VEL
LIN {X 0,Y 240.416,Z 696.137,A -85,B 0,C 180,E1 -19179.252,E2 -19179.252} C_VEL
LIN {X 0,Y 241.151,Z 692.089,A -85,B 0,C 180,E1 -19181.771,E2 -19181.771} C_VEL
LIN {X 0,Y 242.527,Z 685.854,A -85,B 0,C 180,E1 -19184.688,E2 -19184.688} C_VEL
LIN {X 0,Y 244.163,Z 679.056,A -85,B 0,C 180,E1 -19187.16,E2 -19187.16} C_VEL
LIN {X 0,Y 246.119,Z 670.725,A -85,B 0,C 180,E1 -19189.554,E2 -19189.554} C_VEL
LIN {X 0,Y 246.746,Z 668.45,A -85,B 0,C 180,E1 -19190.203,E2 -19190.203} C_VEL
LIN {X 0,Y 249.987,Z 662.368,A -85,B 0,C 180,E1 -19192.741,E2 -19192.741} C_VEL
LIN {X 0,Y 254.356,Z 654.278,A -85,B 0,C 180,E1 -19195.358,E2 -19195.358} C_VEL
LIN {X 0,Y 258.783,Z 645.81,A -85,B 0,C 180,E1 -19197.496,E2 -19197.496} C_VEL
LIN {X 0,Y 263.748,Z 635.7,A -85,B 0,C 180,E1 -19199.536,E2 -19199.536} C_VEL
LIN {X 0,Y 268.378,Z 625.634,A -85,B 0,C 180,E1 -19201.144,E2 -19201.144} C_VEL
LIN {X 0,Y 273.945,Z 612.209,A -85,B 0,C 180,E1 -19202.817,E2 -19202.817} C_VEL
LIN {X 0,Y 278.932,Z 598.522,A -85,B 0,C 180,E1 -19204.098,E2 -19204.098} C_VEL
LIN {X 0,Y 283.33,Z 583.996,A -85,B 0,C 180,E1 -19205.144,E2 -19205.144} C_VEL
LIN {X 0,Y 287.023,Z 568.388,A -85,B 0,C 180,E1 -19205.991,E2 -19205.991} C_VEL
LIN {X 0,Y 291.576,Z 543.007,A -85,B 0,C 180,E1 -19207.183,E2 -19207.183} C_VEL
LIN {X 0,Y 292.602,Z 533.324,A -85,B 0,C 180,E1 -19208.028,E2 -19208.028} C_VEL
LIN {X 0,Y 293.344,Z 523.717,A -85,B 0,C 180,E1 -19209.137,E2 -19209.137} C_VEL
LIN {X 0,Y 293.331,Z 522.313,A -85,B 0,C 180,E1 -19209.397,E2 -19209.397} C_VEL
LIN {X 0,Y 292.815,Z 519.396,A -85,B 0,C 180,E1 -19210.33,E2 -19210.33} C_VEL
LIN {X 0,Y 292.15,Z 515.393,A -85,B 0,C 180,E1 -19211.885,E2 -19211.885} C_VEL
LIN {X 0,Y 291.535,Z 511.609,A -85,B 0,C 180,E1 -19214.355,E2 -19214.355} C_VEL
LIN {X 0,Y 291.638,Z 509.899,A -85,B 0,C 180,E1 -19216.299,E2 -19216.299} C_VEL
LIN {X 0,Y 292.217,Z 509.426,A -85,B 0,C 180,E1 -19218.208,E2 -19218.208} C_VEL
LIN {X 0,Y 293.293,Z 509.515,A -85,B 0,C 180,E1 -19219.935,E2 -19219.935} C_VEL
LIN {X 0,Y 294.955,Z 511.562,A -85,B 0,C 180,E1 -19221.999,E2 -19221.999} C_VEL
LIN {X 0,Y 296.199,Z 513.341,A -85,B 0,C 180,E1 -19223.19,E2 -19223.19} C_VEL
LIN {X 0,Y 290.124,Z 545.411,A -85,B 0,C 180,E1 -19224.718,E2 -19224.718} C_VEL
LIN {X 0,Y 287.612,Z 558.134,A -85,B 0,C 180,E1 -19225.486,E2 -19225.486} C_VEL
LIN {X 0,Y 284.201,Z 571.79,A -85,B 0,C 180,E1 -19226.618,E2 -19226.618} C_VEL
LIN {X 0,Y 280.184,Z 584.61,A -85,B 0,C 180,E1 -19228.002,E2 -19228.002} C_VEL
LIN {X 0,Y 275.841,Z 596.084,A -85,B 0,C 180,E1 -19229.577,E2 -19229.577} C_VEL
LIN {X 0,Y 271.351,Z 606.396,A -85,B 0,C 180,E1 -19231.37,E2 -19231.37} C_VEL
LIN {X 0,Y 266.731,Z 615.582,A -85,B 0,C 180,E1 -19233.389,E2 -19233.389} C_VEL
LIN {X 0,Y 262.611,Z 623.05,A -85,B 0,C 180,E1 -19235.493,E2 -19235.493} C_VEL
LIN {X 0,Y 258.687,Z 629.102,A -85,B 0,C 180,E1 -19237.645,E2 -19237.645} C_VEL
LIN {X 0,Y 255.206,Z 633.983,A -85,B 0,C 180,E1 -19239.865,E2 -19239.865} C_VEL
LIN {X 0,Y 252.016,Z 637.763,A -85,B 0,C 180,E1 -19242.136,E2 -19242.136} C_VEL
LIN {X 0,Y 248.368,Z 641.25,A -85,B 0,C 180,E1 -19245.246,E2 -19245.246} C_VEL
LIN {X 0,Y 246.78,Z 642.375,A -85,B 0,C 180,E1 -19246.831,E2 -19246.831} C_VEL
LIN {X 0,Y 245.388,Z 643.045,A -85,B 0,C 180,E1 -19248.435,E2 -19248.435} C_VEL
LIN {X 0,Y 243.35,Z 643.18,A -85,B 0,C 180,E1 -19251.697,E2 -19251.697} C_VEL
LIN {X 0,Y 242.525,Z 642.658,A -85,B 0,C 180,E1 -19253.344,E2 -19253.344} C_VEL
LIN {X 0,Y 241.281,Z 640.33,A -85,B 0,C 180,E1 -19256.66,E2 -19256.66} C_VEL
LIN {X 0,Y 240.742,Z 637.492,A -85,B 0,C 180,E1 -19259.164,E2 -19259.164} C_VEL
LIN {X 0,Y 240.586,Z 633.619,A -85,B 0,C 180,E1 -19261.674,E2 -19261.674} C_VEL
LIN {X 0,Y 240.775,Z 628.64,A -85,B 0,C 180,E1 -19264.185,E2 -19264.185} C_VEL
LIN {X 0,Y 240.957,Z 622.403,A -85,B 0,C 180,E1 -19266.7,E2 -19266.7} C_VEL
LIN {X 0,Y 241.43,Z 614.71,A -85,B 0,C 180,E1 -19269.213,E2 -19269.213} C_VEL
LIN {X 0,Y 242.112,Z 605.157,A -85,B 0,C 180,E1 -19271.724,E2 -19271.724} C_VEL
LIN {X 0,Y 242.907,Z 595.439,A -85,B 0,C 180,E1 -19273.81,E2 -19273.81} C_VEL
LIN {X 0,Y 243.929,Z 583.478,A -85,B 0,C 180,E1 -19275.885,E2 -19275.885} C_VEL
LIN {X 0,Y 244.855,Z 571.652,A -85,B 0,C 180,E1 -19277.541,E2 -19277.541} C_VEL
LIN {X 0,Y 245.699,Z 558.292,A -85,B 0,C 180,E1 -19279.012,E2 -19279.012} C_VEL
LIN {X 0,Y 246.405,Z 544.971,A -85,B 0,C 180,E1 -19280.124,E2 -19280.124} C_VEL
LIN {X 0,Y 246.951,Z 531.16,A -85,B 0,C 180,E1 -19280.948,E2 -19280.948} C_VEL
LIN {X 0,Y 249.365,Z 468.285,A -85,B 0,C 180,E1 -19283.862,E2 -19283.862} C_VEL
LIN {X 0,Y 242.147,Z 443.729,A -85,B 0,C 180,E1 -19285.344,E2 -19285.344} C_VEL
LIN {X 0,Y 242.086,Z 443.332,A -85,B 0,C 180,E1 -19285.454,E2 -19285.454} C_VEL
LIN {X 0,Y 242.009,Z 443.341,A -85,B 0,C 180,E1 -19289.583,E2 -19289.583} C_VEL
LIN {X 0,Y 241.983,Z 443.308,A -85,B 0,C 180,E1 -19293.493,E2 -19293.493} C_VEL
LIN {X 0,Y 241.993,Z 443.345,A -85,B 0,C 180,E1 -19297.582,E2 -19297.582} C_VEL
LIN {X 0,Y 241.939,Z 443.335,A -85,B 0,C 180,E1 -19301.922,E2 -19301.922} C_VEL
LIN {X 0,Y 241.929,Z 443.334,A -85,B 0,C 180,E1 -19306.573,E2 -19306.573} C_VEL
LIN {X 0,Y 241.98,Z 443.365,A -85,B 0,C 180,E1 -19307.184,E2 -19307.184} C_VEL
LIN {X 0,Y 245.79,Z 454.566,A -85,B 0,C 180,E1 -19311.019,E2 -19311.019} C_VEL
LIN {X 0,Y 248.805,Z 464.629,A -85,B 0,C 180,E1 -19314.157,E2 -19314.157} C_VEL
LIN {X 0,Y 251.334,Z 474.975,A -85,B 0,C 180,E1 -19317.087,E2 -19317.087} C_VEL
LIN {X 0,Y 257.053,Z 488.252,A -85,B 0,C 180,E1 -19318.341,E2 -19318.341} C_VEL
LIN {X 0,Y 261.026,Z 512.484,A -85,B 0,C 180,E1 -19319.643,E2 -19319.643} C_VEL
LIN {X 0,Y 261.011,Z 519.344,A -85,B 0,C 180,E1 -19319.856,E2 -19319.856} C_VEL
LIN {X 0,Y 258.715,Z 582.857,A -85,B 0,C 180,E1 -19321.56,E2 -19321.56} C_VEL
LIN {X 0,Y 257.885,Z 596.008,A -85,B 0,C 180,E1 -19322.124,E2 -19322.124} C_VEL
LIN {X 0,Y 256.584,Z 608.067,A -85,B 0,C 180,E1 -19322.911,E2 -19322.911} C_VEL
LIN {X 0,Y 254.958,Z 620.404,A -85,B 0,C 180,E1 -19324.049,E2 -19324.049} C_VEL
LIN {X 0,Y 253.086,Z 631.368,A -85,B 0,C 180,E1 -19325.384,E2 -19325.384} C_VEL
LIN {X 0,Y 250.856,Z 642.667,A -85,B 0,C 180,E1 -19327.147,E2 -19327.147} C_VEL
LIN {X 0,Y 248.819,Z 652.303,A -85,B 0,C 180,E1 -19329.066,E2 -19329.066} C_VEL
LIN {X 0,Y 246.649,Z 661.296,A -85,B 0,C 180,E1 -19331.303,E2 -19331.303} C_VEL
LIN {X 0,Y 244.592,Z 669.091,A -85,B 0,C 180,E1 -19333.731,E2 -19333.731} C_VEL
LIN {X 0,Y 243.299,Z 674.351,A -85,B 0,C 180,E1 -19335.787,E2 -19335.787} C_VEL
LIN {X 0,Y 241.962,Z 679.49,A -85,B 0,C 180,E1 -19338.269,E2 -19338.269} C_VEL
LIN {X 0,Y 241.033,Z 683.465,A -85,B 0,C 180,E1 -19340.772,E2 -19340.772} C_VEL
LIN {X 0,Y 240.302,Z 686.971,A -85,B 0,C 180,E1 -19343.926,E2 -19343.926} C_VEL
LIN {X 0,Y 240.008,Z 688.803,A -85,B 0,C 180,E1 -19346.643,E2 -19346.643} C_VEL
LIN {X 0,Y 239.913,Z 689.415,A -85,B 0,C 180,E1 -19348.321,E2 -19348.321} C_VEL
LIN {X 0,Y 239.893,Z 689.647,A -85,B 0,C 180,E1 -19350,E2 -19350} C_VEL
LIN {X 0,Y 239.912,Z 689.451,A -85,B 0,C 180,E1 -19351.679,E2 -19351.679} C_VEL
LIN {X 0,Y 240.008,Z 688.862,A -85,B 0,C 180,E1 -19353.357,E2 -19353.357} C_VEL
LIN {X 0,Y 240.319,Z 687.045,A -85,B 0,C 180,E1 -19356.11,E2 -19356.11} C_VEL
LIN {X 0,Y 241.013,Z 683.641,A -85,B 0,C 180,E1 -19359.229,E2 -19359.229} C_VEL
LIN {X 0,Y 241.924,Z 679.725,A -85,B 0,C 180,E1 -19361.733,E2 -19361.733} C_VEL
LIN {X 0,Y 243.254,Z 674.645,A -85,B 0,C 180,E1 -19364.216,E2 -19364.216} C_VEL
LIN {X 0,Y 244.871,Z 668.241,A -85,B 0,C 180,E1 -19366.679,E2 -19366.679} C_VEL
LIN {X 0,Y 246.999,Z 660.277,A -85,B 0,C 180,E1 -19369.1,E2 -19369.1} C_VEL
LIN {X 0,Y 248.935,Z 652.037,A -85,B 0,C 180,E1 -19371.122,E2 -19371.122} C_VEL
LIN {X 0,Y 251.004,Z 642.101,A -85,B 0,C 180,E1 -19373.079,E2 -19373.079} C_VEL
LIN {X 0,Y 253.289,Z 630.81,A -85,B 0,C 180,E1 -19374.814,E2 -19374.814} C_VEL
LIN {X 0,Y 255.11,Z 619.688,A -85,B 0,C 180,E1 -19376.154,E2 -19376.154} C_VEL
LIN {X 0,Y 256.862,Z 607.071,A -85,B 0,C 180,E1 -19377.277,E2 -19377.277} C_VEL
LIN {X 0,Y 258.016,Z 594.635,A -85,B 0,C 180,E1 -19378.081,E2 -19378.081} C_VEL
LIN {X 0,Y 258.853,Z 581.823,A -85,B 0,C 180,E1 -19378.589,E2 -19378.589} C_VEL
LIN {X 0,Y 261.277,Z 513.899,A -85,B 0,C 180,E1 -19380.412,E2 -19380.412} C_VEL
LIN {X 0,Y 257.301,Z 489.569,A -85,B 0,C 180,E1 -19381.716,E2 -19381.716} C_VEL
LIN {X 0,Y 256.359,Z 486.352,A -85,B 0,C 180,E1 -19381.951,E2 -19381.951} C_VEL
LIN {X 0,Y 251.365,Z 474.8,A -85,B 0,C 180,E1 -19383.082,E2 -19383.082} C_VEL
LIN {X 0,Y 248.189,Z 462.513,A -85,B 0,C 180,E1 -19386.627,E2 -19386.627} C_VEL
LIN {X 0,Y 245.256,Z 452.933,A -85,B 0,C 180,E1 -19389.699,E2 -19389.699} C_VEL
LIN {X 0,Y 241.971,Z 443.337,A -85,B 0,C 180,E1 -19393.004,E2 -19393.004} C_VEL
LIN {X 0,Y 241.939,Z 443.347,A -85,B 0,C 180,E1 -19396.57,E2 -19396.57} C_VEL
LIN {X 0,Y 241.959,Z 443.347,A -85,B 0,C 180,E1 -19400.281,E2 -19400.281} C_VEL
LIN {X 0,Y 242.006,Z 443.321,A -85,B 0,C 180,E1 -19404.492,E2 -19404.492} C_VEL
LIN {X 0,Y 242.049,Z 443.415,A -85,B 0,C 180,E1 -19405.892,E2 -19405.892} C_VEL
LIN {X 0,Y 245.382,Z 459.15,A -85,B 0,C 180,E1 -19409.999,E2 -19409.999} C_VEL
LIN {X 0,Y 247.216,Z 468.16,A -85,B 0,C 180,E1 -19412.296,E2 -19412.296} C_VEL
LIN {X 0,Y 246.833,Z 474.568,A -85,B 0,C 180,E1 -19413.811,E2 -19413.811} C_VEL
LIN {X 0,Y 246.735,Z 475.492,A -85,B 0,C 180,E1 -19414.027,E2 -19414.027} C_VEL
LIN {X 0,Y 248.562,Z 497.484,A -85,B 0,C 180,E1 -19415.174,E2 -19415.174} C_VEL
LIN {X 0,Y 249.378,Z 504.404,A -85,B 0,C 180,E1 -19415.535,E2 -19415.535} C_VEL
LIN {X 0,Y 249.368,Z 508.235,A -85,B 0,C 180,E1 -19415.713,E2 -19415.713} C_VEL
LIN {X 0,Y 248.143,Z 513.934,A -85,B 0,C 180,E1 -19415.933,E2 -19415.933} C_VEL
LIN {X 0,Y 242.621,Z 528.833,A -85,B 0,C 180,E1 -19416.463,E2 -19416.463} C_VEL
LIN {X 0,Y 241.634,Z 534.643,A -85,B 0,C 180,E1 -19416.719,E2 -19416.719} C_VEL
LIN {X 0,Y 239.4,Z 587.654,A -85,B 0,C 180,E1 -19419.317,E2 -19419.317} C_VEL
LIN {X 0,Y 238.565,Z 602.518,A -85,B 0,C 180,E1 -19420.398,E2 -19420.398} C_VEL
LIN {X 0,Y 237.606,Z 615.365,A -85,B 0,C 180,E1 -19421.683,E2 -19421.683} C_VEL
LIN {X 0,Y 236.675,Z 627.063,A -85,B 0,C 180,E1 -19423.17,E2 -19423.17} C_VEL
LIN {X 0,Y 235.885,Z 636.638,A -85,B 0,C 180,E1 -19424.667,E2 -19424.667} C_VEL
LIN {X 0,Y 234.895,Z 647.874,A -85,B 0,C 180,E1 -19426.812,E2 -19426.812} C_VEL
LIN {X 0,Y 234.218,Z 656.192,A -85,B 0,C 180,E1 -19428.753,E2 -19428.753} C_VEL
LIN {X 0,Y 233.565,Z 665.271,A -85,B 0,C 180,E1 -19431.347,E2 -19431.347} C_VEL
LIN {X 0,Y 233.137,Z 671.995,A -85,B 0,C 180,E1 -19433.704,E2 -19433.704} C_VEL
LIN {X 0,Y 232.979,Z 678.482,A -85,B 0,C 180,E1 -19436.541,E2 -19436.541} C_VEL
LIN {X 0,Y 232.832,Z 683.05,A -85,B 0,C 180,E1 -19439.135,E2 -19439.135} C_VEL
LIN {X 0,Y 232.907,Z 686.471,A -85,B 0,C 180,E1 -19441.729,E2 -19441.729} C_VEL
LIN {X 0,Y 233.192,Z 689.486,A -85,B 0,C 180,E1 -19445.187,E2 -19445.187} C_VEL
LIN {X 0,Y 233.593,Z 690.341,A -85,B 0,C 180,E1 -19446.912,E2 -19446.912} C_VEL
LIN {X 0,Y 234.907,Z 690.876,A -85,B 0,C 180,E1 -19450.341,E2 -19450.341} C_VEL
LIN {X 0,Y 235.888,Z 690.542,A -85,B 0,C 180,E1 -19452.038,E2 -19452.038} C_VEL
LIN {X 0,Y 238.399,Z 688.63,A -85,B 0,C 180,E1 -19455.386,E2 -19455.386} C_VEL
LIN {X 0,Y 239.857,Z 687.131,A -85,B 0,C 180,E1 -19457.038,E2 -19457.038} C_VEL
LIN {X 0,Y 242.853,Z 683.979,A -85,B 0,C 180,E1 -19459.439,E2 -19459.439} C_VEL
LIN {X 0,Y 246.074,Z 679.836,A -85,B 0,C 180,E1 -19461.795,E2 -19461.795} C_VEL
LIN {X 0,Y 250.508,Z 673.616,A -85,B 0,C 180,E1 -19464.445,E2 -19464.445} C_VEL
LIN {X 0,Y 255.552,Z 665.687,A -85,B 0,C 180,E1 -19466.986,E2 -19466.986} C_VEL
LIN {X 0,Y 260.344,Z 657.259,A -85,B 0,C 180,E1 -19469.072,E2 -19469.072} C_VEL
LIN {X 0,Y 265.546,Z 647.003,A -85,B 0,C 180,E1 -19471.071,E2 -19471.071} C_VEL
LIN {X 0,Y 270.191,Z 636.637,A -85,B 0,C 180,E1 -19472.665,E2 -19472.665} C_VEL
LIN {X 0,Y 274.644,Z 625.273,A -85,B 0,C 180,E1 -19474.04,E2 -19474.04} C_VEL
LIN {X 0,Y 278.816,Z 612.915,A -85,B 0,C 180,E1 -19475.212,E2 -19475.212} C_VEL
LIN {X 0,Y 282.355,Z 600.045,A -85,B 0,C 180,E1 -19476.128,E2 -19476.128} C_VEL
LIN {X 0,Y 286.116,Z 582.713,A -85,B 0,C 180,E1 -19476.999,E2 -19476.999} C_VEL
LIN {X 0,Y 295.725,Z 535.279,A -85,B 0,C 180,E1 -19479.132,E2 -19479.132} C_VEL
LIN {X 0,Y 295.19,Z 532.403,A -85,B 0,C 180,E1 -19480.225,E2 -19480.225} C_VEL
LIN {X 0,Y 294.728,Z 529.979,A -85,B 0,C 180,E1 -19481.487,E2 -19481.487} C_VEL
LIN {X 0,Y 294.226,Z 527.388,A -85,B 0,C 180,E1 -19483.733,E2 -19483.733} C_VEL
LIN {X 0,Y 294.3,Z 526.781,A -85,B 0,C 180,E1 -19485.759,E2 -19485.759} C_VEL
LIN {X 0,Y 295.261,Z 527.364,A -85,B 0,C 180,E1 -19488.204,E2 -19488.204} C_VEL
LIN {X 0,Y 296.039,Z 528.315,A -85,B 0,C 180,E1 -19489.437,E2 -19489.437} C_VEL
LIN {X 0,Y 294.441,Z 539.101,A -85,B 0,C 180,E1 -19490.587,E2 -19490.587} C_VEL
LIN {X 0,Y 293.31,Z 545.969,A -85,B 0,C 180,E1 -19491.146,E2 -19491.146} C_VEL
LIN {X 0,Y 291.954,Z 552.844,A -85,B 0,C 180,E1 -19491.492,E2 -19491.492} C_VEL
LIN {X 0,Y 281.622,Z 603.511,A -85,B 0,C 180,E1 -19493.873,E2 -19493.873} C_VEL
LIN {X 0,Y 278.007,Z 616.639,A -85,B 0,C 180,E1 -19494.67,E2 -19494.67} C_VEL
LIN {X 0,Y 273.477,Z 630.099,A -85,B 0,C 180,E1 -19495.779,E2 -19495.779} C_VEL
LIN {X 0,Y 269.701,Z 639.913,A -85,B 0,C 180,E1 -19496.823,E2 -19496.823} C_VEL
LIN {X 0,Y 264.654,Z 651.323,A -85,B 0,C 180,E1 -19498.367,E2 -19498.367} C_VEL
LIN {X 0,Y 260.022,Z 660.916,A -85,B 0,C 180,E1 -19499.998,E2 -19499.998} C_VEL
LIN {X 0,Y 255.746,Z 668.924,A -85,B 0,C 180,E1 -19501.703,E2 -19501.703} C_VEL
LIN {X 0,Y 250.909,Z 677.367,A -85,B 0,C 180,E1 -19503.958,E2 -19503.958} C_VEL
LIN {X 0,Y 246.348,Z 684.629,A -85,B 0,C 180,E1 -19506.459,E2 -19506.459} C_VEL
LIN {X 0,Y 242.855,Z 689.894,A -85,B 0,C 180,E1 -19508.793,E2 -19508.793} C_VEL
LIN {X 0,Y 239.763,Z 694.049,A -85,B 0,C 180,E1 -19511.19,E2 -19511.19} C_VEL
LIN {X 0,Y 238.146,Z 696.258,A -85,B 0,C 180,E1 -19512.836,E2 -19512.836} C_VEL
LIN {X 0,Y 235.58,Z 699.429,A -85,B 0,C 180,E1 -19516.192,E2 -19516.192} C_VEL
LIN {X 0,Y 234.596,Z 700.435,A -85,B 0,C 180,E1 -19517.895,E2 -19517.895} C_VEL
LIN {X 0,Y 233.876,Z 701.012,A -85,B 0,C 180,E1 -19519.613,E2 -19519.613} C_VEL
LIN {X 0,Y 232.994,Z 700.973,A -85,B 0,C 180,E1 -19523.07,E2 -19523.07} C_VEL
LIN {X 0,Y 232.881,Z 700.399,A -85,B 0,C 180,E1 -19524.806,E2 -19524.806} C_VEL
LIN {X 0,Y 232.82,Z 702.022,A -85,B 0,C 180,E1 -19528.27,E2 -19528.27} C_VEL
LIN {X 0,Y 232.863,Z 702.239,A -85,B 0,C 180,E1 -19530,E2 -19530} C_VEL
LIN {X 0,Y 232.788,Z 702.01,A -85,B 0,C 180,E1 -19531.73,E2 -19531.73} C_VEL
LIN {X 0,Y 232.763,Z 700.589,A -85,B 0,C 180,E1 -19534.864,E2 -19534.864} C_VEL
LIN {X 0,Y 232.917,Z 698.933,A -85,B 0,C 180,E1 -19536.932,E2 -19536.932} C_VEL
LIN {X 0,Y 233.391,Z 695.948,A -85,B 0,C 180,E1 -19539.533,E2 -19539.533} C_VEL
LIN {X 0,Y 234.162,Z 691.898,A -85,B 0,C 180,E1 -19542.128,E2 -19542.128} C_VEL
LIN {X 0,Y 235.644,Z 685.664,A -85,B 0,C 180,E1 -19545.127,E2 -19545.127} C_VEL
LIN {X 0,Y 237.342,Z 678.867,A -85,B 0,C 180,E1 -19547.669,E2 -19547.669} C_VEL
LIN {X 0,Y 239.255,Z 671.215,A -85,B 0,C 180,E1 -19549.951,E2 -19549.951} C_VEL
LIN {X 0,Y 239.746,Z 669.476,A -85,B 0,C 180,E1 -19550.461,E2 -19550.461} C_VEL
LIN {X 0,Y 242.936,Z 664.108,A -85,B 0,C 180,E1 -19552.989,E2 -19552.989} C_VEL
LIN {X 0,Y 246.683,Z 657.884,A -85,B 0,C 180,E1 -19555.3,E2 -19555.3} C_VEL
LIN {X 0,Y 251.047,Z 650.432,A -85,B 0,C 180,E1 -19557.511,E2 -19557.511} C_VEL
LIN {X 0,Y 256.014,Z 641.508,A -85,B 0,C 180,E1 -19559.612,E2 -19559.612} C_VEL
LIN {X 0,Y 261.525,Z 630.799,A -85,B 0,C 180,E1 -19561.603,E2 -19561.603} C_VEL
LIN {X 0,Y 266.707,Z 620.067,A -85,B 0,C 180,E1 -19563.147,E2 -19563.147} C_VEL
LIN {X 0,Y 271.574,Z 608.573,A -85,B 0,C 180,E1 -19564.479,E2 -19564.479} C_VEL
LIN {X 0,Y 276.809,Z 594.542,A -85,B 0,C 180,E1 -19565.729,E2 -19565.729} C_VEL
LIN {X 0,Y 281.306,Z 580.138,A -85,B 0,C 180,E1 -19566.674,E2 -19566.674} C_VEL
LIN {X 0,Y 285.12,Z 563.906,A -85,B 0,C 180,E1 -19567.532,E2 -19567.532} C_VEL
LIN {X 0,Y 288.831,Z 544.473,A -85,B 0,C 180,E1 -19568.448,E2 -19568.448} C_VEL
LIN {X 0,Y 289.973,Z 535.449,A -85,B 0,C 180,E1 -19569.262,E2 -19569.262} C_VEL
LIN {X 0,Y 290.786,Z 527.448,A -85,B 0,C 180,E1 -19570.222,E2 -19570.222} C_VEL
LIN {X 0,Y 290.089,Z 521.889,A -85,B 0,C 180,E1 -19572.275,E2 -19572.275} C_VEL
LIN {X 0,Y 289.657,Z 518.205,A -85,B 0,C 180,E1 -19574.719,E2 -19574.719} C_VEL
LIN {X 0,Y 289.878,Z 516.623,A -85,B 0,C 180,E1 -19576.664,E2 -19576.664} C_VEL
LIN {X 0,Y 291.022,Z 516.255,A -85,B 0,C 180,E1 -19579.305,E2 -19579.305} C_VEL
LIN {X 0,Y 291.835,Z 516.944,A -85,B 0,C 180,E1 -19580.535,E2 -19580.535} C_VEL
LIN {X 0,Y 293.156,Z 518.705,A -85,B 0,C 180,E1 -19582.098,E2 -19582.098} C_VEL
LIN {X 0,Y 287.534,Z 546.506,A -85,B 0,C 180,E1 -19583.426,E2 -19583.426} C_VEL
LIN {X 0,Y 284.749,Z 559.592,A -85,B 0,C 180,E1 -19584.222,E2 -19584.222} C_VEL
LIN {X 0,Y 281.133,Z 572.96,A -85,B 0,C 180,E1 -19585.339,E2 -19585.339} C_VEL
LIN {X 0,Y 276.869,Z 585.596,A -85,B 0,C 180,E1 -19586.707,E2 -19586.707} C_VEL
LIN {X 0,Y 272.263,Z 596.96,A -85,B 0,C 180,E1 -19588.268,E2 -19588.268} C_VEL
LIN {X 0,Y 267.463,Z 607.219,A -85,B 0,C 180,E1 -19590.049,E2 -19590.049} C_VEL
LIN {X 0,Y 262.761,Z 615.928,A -85,B 0,C 180,E1 -19591.963,E2 -19591.963} C_VEL
LIN {X 0,Y 258.034,Z 623.778,A -85,B 0,C 180,E1 -19594.165,E2 -19594.165} C_VEL
LIN {X 0,Y 253.817,Z 629.93,A -85,B 0,C 180,E1 -19596.328,E2 -19596.328} C_VEL
LIN {X 0,Y 250.034,Z 634.768,A -85,B 0,C 180,E1 -19598.567,E2 -19598.567} C_VEL
LIN {X 0,Y 245.507,Z 639.609,A -85,B 0,C 180,E1 -19601.646,E2 -19601.646} C_VEL
LIN {X 0,Y 243.485,Z 641.392,A -85,B 0,C 180,E1 -19603.223,E2 -19603.223} C_VEL
LIN {X 0,Y 239.98,Z 643.619,A -85,B 0,C 180,E1 -19606.45,E2 -19606.45} C_VEL
LIN {X 0,Y 238.538,Z 644.151,A -85,B 0,C 180,E1 -19608.098,E2 -19608.098} C_VEL
LIN {X 0,Y 237.375,Z 644.266,A -85,B 0,C 180,E1 -19609.768,E2 -19609.768} C_VEL
LIN {X 0,Y 235.516,Z 643.239,A -85,B 0,C 180,E1 -19613.145,E2 -19613.145} C_VEL
LIN {X 0,Y 234.802,Z 642.14,A -85,B 0,C 180,E1 -19614.848,E2 -19614.848} C_VEL
LIN {X 0,Y 234.201,Z 640.635,A -85,B 0,C 180,E1 -19616.559,E2 -19616.559} C_VEL
LIN {X 0,Y 233.642,Z 637.545,A -85,B 0,C 180,E1 -19619.138,E2 -19619.138} C_VEL
LIN {X 0,Y 233.497,Z 633.442,A -85,B 0,C 180,E1 -19621.725,E2 -19621.725} C_VEL
LIN {X 0,Y 233.774,Z 627.18,A -85,B 0,C 180,E1 -19624.742,E2 -19624.742} C_VEL
LIN {X 0,Y 233.973,Z 619.65,A -85,B 0,C 180,E1 -19627.586,E2 -19627.586} C_VEL
LIN {X 0,Y 234.479,Z 612.015,A -85,B 0,C 180,E1 -19629.924,E2 -19629.924} C_VEL
LIN {X 0,Y 235.297,Z 601.672,A -85,B 0,C 180,E1 -19632.506,E2 -19632.506} C_VEL
LIN {X 0,Y 236.154,Z 591.096,A -85,B 0,C 180,E1 -19634.653,E2 -19634.653} C_VEL
LIN {X 0,Y 237.115,Z 579.391,A -85,B 0,C 180,E1 -19636.576,E2 -19636.576} C_VEL
LIN {X 0,Y 238.022,Z 568.195,A -85,B 0,C 180,E1 -19638.061,E2 -19638.061} C_VEL
LIN {X 0,Y 238.796,Z 554.58,A -85,B 0,C 180,E1 -19639.477,E2 -19639.477} C_VEL
LIN {X 0,Y 239.612,Z 540.369,A -85,B 0,C 180,E1 -19640.57,E2 -19640.57} C_VEL
LIN {X 0,Y 240.319,Z 518.071,A -85,B 0,C 180,E1 -19641.723,E2 -19641.723} C_VEL
LIN {X 0,Y 242.321,Z 469.363,A -85,B 0,C 180,E1 -19644.071,E2 -19644.071} C_VEL
LIN {X 0,Y 235.457,Z 445.969,A -85,B 0,C 180,E1 -19645.527,E2 -19645.527} C_VEL
LIN {X 0,Y 235.042,Z 444.208,A -85,B 0,C 180,E1 -19645.69,E2 -19645.69} C_VEL
LIN {X 0,Y 234.924,Z 444.22,A -85,B 0,C 180,E1 -19650.569,E2 -19650.569} C_VEL
LIN {X 0,Y 234.933,Z 444.189,A -85,B 0,C 180,E1 -19654.638,E2 -19654.638} C_VEL
LIN {X 0,Y 234.944,Z 444.206,A -85,B 0,C 180,E1 -19658.944,E2 -19658.944} C_VEL
LIN {X 0,Y 234.887,Z 444.232,A -85,B 0,C 180,E1 -19663.486,E2 -19663.486} C_VEL
LIN {X 0,Y 234.889,Z 444.247,A -85,B 0,C 180,E1 -19665.897,E2 -19665.897} C_VEL
LIN {X 0,Y 238.821,Z 455.47,A -85,B 0,C 180,E1 -19669.919,E2 -19669.919} C_VEL
LIN {X 0,Y 241.309,Z 463.343,A -85,B 0,C 180,E1 -19672.526,E2 -19672.526} C_VEL
LIN {X 0,Y 244.342,Z 474.907,A -85,B 0,C 180,E1 -19675.969,E2 -19675.969} C_VEL
LIN {X 0,Y 250.472,Z 488.942,A -85,B 0,C 180,E1 -19677.428,E2 -19677.428} C_VEL
LIN {X 0,Y 251.542,Z 492.342,A -85,B 0,C 180,E1 -19677.697,E2 -19677.697} C_VEL
LIN {X 0,Y 255.045,Z 514.554,A -85,B 0,C 180,E1 -19678.916,E2 -19678.916} C_VEL
LIN {X 0,Y 252.452,Z 584.344,A -85,B 0,C 180,E1 -19680.844,E2 -19680.844} C_VEL
LIN {X 0,Y 251.447,Z 597.858,A -85,B 0,C 180,E1 -19681.46,E2 -19681.46} C_VEL
LIN {X 0,Y 250.15,Z 609.465,A -85,B 0,C 180,E1 -19682.269,E2 -19682.269} C_VEL
LIN {X 0,Y 248.612,Z 620.58,A -85,B 0,C 180,E1 -19683.335,E2 -19683.335} C_VEL
LIN {X 0,Y 246.649,Z 631.548,A -85,B 0,C 180,E1 -19684.697,E2 -19684.697} C_VEL
LIN {X 0,Y 244.341,Z 642.85,A -85,B 0,C 180,E1 -19686.501,E2 -19686.501} C_VEL
LIN {X 0,Y 242.078,Z 652.934,A -85,B 0,C 180,E1 -19688.568,E2 -19688.568} C_VEL
LIN {X 0,Y 239.941,Z 661.483,A -85,B 0,C 180,E1 -19690.76,E2 -19690.76} C_VEL
LIN {X 0,Y 237.786,Z 669.279,A -85,B 0,C 180,E1 -19693.251,E2 -19693.251} C_VEL
LIN {X 0,Y 236.417,Z 674.539,A -85,B 0,C 180,E1 -19695.364,E2 -19695.364} C_VEL
LIN {X 0,Y 235.013,Z 679.679,A -85,B 0,C 180,E1 -19697.917,E2 -19697.917} C_VEL
LIN {X 0,Y 234.027,Z 683.654,A -85,B 0,C 180,E1 -19700.493,E2 -19700.493} C_VEL
LIN {X 0,Y 233.226,Z 687.328,A -85,B 0,C 180,E1 -19703.947,E2 -19703.947} C_VEL
LIN {X 0,Y 232.915,Z 688.993,A -85,B 0,C 180,E1 -19706.54,E2 -19706.54} C_VEL
LIN {X 0,Y 232.828,Z 689.604,A -85,B 0,C 180,E1 -19708.27,E2 -19708.27} C_VEL
LIN {X 0,Y 232.805,Z 689.836,A -85,B 0,C 180,E1 -19710,E2 -19710} C_VEL
LIN {X 0,Y 232.828,Z 689.639,A -85,B 0,C 180,E1 -19711.73,E2 -19711.73} C_VEL
LIN {X 0,Y 232.915,Z 689.051,A -85,B 0,C 180,E1 -19713.46,E2 -19713.46} C_VEL
LIN {X 0,Y 233.236,Z 687.413,A -85,B 0,C 180,E1 -19716.076,E2 -19716.076} C_VEL
LIN {X 0,Y 234.008,Z 683.828,A -85,B 0,C 180,E1 -19719.508,E2 -19719.508} C_VEL
LIN {X 0,Y 234.979,Z 679.911,A -85,B 0,C 180,E1 -19722.085,E2 -19722.085} C_VEL
LIN {X 0,Y 236.377,Z 674.83,A -85,B 0,C 180,E1 -19724.639,E2 -19724.639} C_VEL
LIN {X 0,Y 238.076,Z 668.425,A -85,B 0,C 180,E1 -19727.17,E2 -19727.17} C_VEL
LIN {X 0,Y 240.307,Z 660.459,A -85,B 0,C 180,E1 -19729.653,E2 -19729.653} C_VEL
LIN {X 0,Y 242.454,Z 651.683,A -85,B 0,C 180,E1 -19731.848,E2 -19731.848} C_VEL
LIN {X 0,Y 244.495,Z 642.277,A -85,B 0,C 180,E1 -19733.73,E2 -19733.73} C_VEL
LIN {X 0,Y 246.864,Z 630.981,A -85,B 0,C 180,E1 -19735.505,E2 -19735.505} C_VEL
LIN {X 0,Y 248.765,Z 619.851,A -85,B 0,C 180,E1 -19736.874,E2 -19736.874} C_VEL
LIN {X 0,Y 250.585,Z 607.22,A -85,B 0,C 180,E1 -19738.02,E2 -19738.02} C_VEL
LIN {X 0,Y 251.794,Z 594.765,A -85,B 0,C 180,E1 -19738.839,E2 -19738.839} C_VEL
LIN {X 0,Y 252.66,Z 581.889,A -85,B 0,C 180,E1 -19739.358,E2 -19739.358} C_VEL
LIN {X 0,Y 255.117,Z 514.631,A -85,B 0,C 180,E1 -19741.206,E2 -19741.206} C_VEL
LIN {X 0,Y 251.432,Z 491.712,A -85,B 0,C 180,E1 -19742.477,E2 -19742.477} C_VEL
LIN {X 0,Y 250.076,Z 487.824,A -85,B 0,C 180,E1 -19742.805,E2 -19742.805} C_VEL
LIN {X 0,Y 244.37,Z 475.078,A -85,B 0,C 180,E1 -19744.133,E2 -19744.133} C_VEL
LIN {X 0,Y 241.445,Z 463.672,A -85,B 0,C 180,E1 -19747.516,E2 -19747.516} C_VEL
LIN {X 0,Y 238.466,Z 454.262,A -85,B 0,C 180,E1 -19750.665,E2 -19750.665} C_VEL
LIN {X 0,Y 234.892,Z 444.217,A -85,B 0,C 180,E1 -19754.349,E2 -19754.349} C_VEL
LIN {X 0,Y 234.886,Z 444.213,A -85,B 0,C 180,E1 -19758.832,E2 -19758.832} C_VEL
LIN {X 0,Y 234.921,Z 444.224,A -85,B 0,C 180,E1 -19761.079,E2 -19761.079} C_VEL
LIN {X 0,Y 235.003,Z 444.256,A -85,B 0,C 180,E1 -19765.584,E2 -19765.584} C_VEL
LIN {X 0,Y 238.199,Z 459.373,A -85,B 0,C 180,E1 -19769.616,E2 -19769.616} C_VEL
LIN {X 0,Y 240.136,Z 468.871,A -85,B 0,C 180,E1 -19772.078,E2 -19772.078} C_VEL
LIN {X 0,Y 240.08,Z 472.74,A -85,B 0,C 180,E1 -19773.016,E2 -19773.016} C_VEL
LIN {X 0,Y 239.765,Z 475.759,A -85,B 0,C 180,E1 -19773.741,E2 -19773.741} C_VEL
LIN {X 0,Y 241.576,Z 498.119,A -85,B 0,C 180,E1 -19774.919,E2 -19774.919} C_VEL
LIN {X 0,Y 242.807,Z 509.6,A -85,B 0,C 180,E1 -19775.527,E2 -19775.527} C_VEL
LIN {X 0,Y 241.634,Z 534.643,A -85,B 0,C 180,E1 -19776.719,E2 -19776.719} C_VEL
LIN {X 0,Y 240.726,Z 540.377,A -85,B 0,C 180,E1 -19776.976,E2 -19776.976} C_VEL
LIN {X 0,Y 234.204,Z 558.841,A -85,B 0,C 180,E1 -19777.735,E2 -19777.735} C_VEL
LIN {X 0,Y 233.293,Z 564.571,A -85,B 0,C 180,E1 -19778.011,E2 -19778.011} C_VEL
LIN {X 0,Y 232.139,Z 590.445,A -85,B 0,C 180,E1 -19779.394,E2 -19779.394} C_VEL
LIN {X 0,Y 231.344,Z 604.196,A -85,B 0,C 180,E1 -19780.478,E2 -19780.478} C_VEL
LIN {X 0,Y 230.439,Z 616.669,A -85,B 0,C 180,E1 -19781.805,E2 -19781.805} C_VEL
LIN {X 0,Y 229.474,Z 629.35,A -85,B 0,C 180,E1 -19783.543,E2 -19783.543} C_VEL
LIN {X 0,Y 228.449,Z 640.889,A -85,B 0,C 180,E1 -19785.525,E2 -19785.525} C_VEL
LIN {X 0,Y 227.431,Z 652.21,A -85,B 0,C 180,E1 -19787.96,E2 -19787.96} C_VEL
LIN {X 0,Y 226.688,Z 662.138,A -85,B 0,C 180,E1 -19790.632,E2 -19790.632} C_VEL
LIN {X 0,Y 226.151,Z 670.152,A -85,B 0,C 180,E1 -19793.308,E2 -19793.308} C_VEL
LIN {X 0,Y 225.921,Z 677.478,A -85,B 0,C 180,E1 -19796.433,E2 -19796.433} C_VEL
LIN {X 0,Y 225.769,Z 682.294,A -85,B 0,C 180,E1 -19799.108,E2 -19799.108} C_VEL
LIN {X 0,Y 225.843,Z 685.978,A -85,B 0,C 180,E1 -19801.783,E2 -19801.783} C_VEL
LIN {X 0,Y 225.899,Z 687.839,A -85,B 0,C 180,E1 -19803.567,E2 -19803.567} C_VEL
LIN {X 0,Y 226.419,Z 690.065,A -85,B 0,C 180,E1 -19806.647,E2 -19806.647} C_VEL
LIN {X 0,Y 227.169,Z 690.951,A -85,B 0,C 180,E1 -19808.899,E2 -19808.899} C_VEL
LIN {X 0,Y 228.966,Z 690.984,A -85,B 0,C 180,E1 -19812.407,E2 -19812.407} C_VEL
LIN {X 0,Y 231.611,Z 689.491,A -85,B 0,C 180,E1 -19815.849,E2 -19815.849} C_VEL
LIN {X 0,Y 233.161,Z 688.132,A -85,B 0,C 180,E1 -19817.543,E2 -19817.543} C_VEL
LIN {X 0,Y 237.345,Z 684.162,A -85,B 0,C 180,E1 -19820.814,E2 -19820.814} C_VEL
LIN {X 0,Y 240.931,Z 680.036,A -85,B 0,C 180,E1 -19823.191,E2 -19823.191} C_VEL
LIN {X 0,Y 246.496,Z 672.806,A -85,B 0,C 180,E1 -19826.227,E2 -19826.227} C_VEL
LIN {X 0,Y 251.217,Z 665.919,A -85,B 0,C 180,E1 -19828.398,E2 -19828.398} C_VEL
LIN {X 0,Y 257.219,Z 656.046,A -85,B 0,C 180,E1 -19830.818,E2 -19830.818} C_VEL
LIN {X 0,Y 262.819,Z 645.475,A -85,B 0,C 180,E1 -19832.786,E2 -19832.786} C_VEL
LIN {X 0,Y 267.862,Z 634.872,A -85,B 0,C 180,E1 -19834.34,E2 -19834.34} C_VEL
LIN {X 0,Y 272.559,Z 623.178,A -85,B 0,C 180,E1 -19835.689,E2 -19835.689} C_VEL
LIN {X 0,Y 277.033,Z 610.316,A -85,B 0,C 180,E1 -19836.823,E2 -19836.823} C_VEL
LIN {X 0,Y 280.551,Z 597.969,A -85,B 0,C 180,E1 -19837.634,E2 -19837.634} C_VEL
LIN {X 0,Y 290.62,Z 551.44,A -85,B 0,C 180,E1 -19839.781,E2 -19839.781} C_VEL
LIN {X 0,Y 293.172,Z 539.521,A -85,B 0,C 180,E1 -19840.335,E2 -19840.335} C_VEL
LIN {X 0,Y 292.746,Z 536.646,A -85,B 0,C 180,E1 -19841.766,E2 -19841.766} C_VEL
LIN {X 0,Y 292.4,Z 534.144,A -85,B 0,C 180,E1 -19843.972,E2 -19843.972} C_VEL
LIN {X 0,Y 292.6,Z 533.636,A -85,B 0,C 180,E1 -19846.102,E2 -19846.102} C_VEL
LIN {X 0,Y 293.445,Z 534.238,A -85,B 0,C 180,E1 -19848.197,E2 -19848.197} C_VEL
LIN {X 0,Y 293.621,Z 534.853,A -85,B 0,C 180,E1 -19848.661,E2 -19848.661} C_VEL
LIN {X 0,Y 291.833,Z 544.953,A -85,B 0,C 180,E1 -19849.659,E2 -19849.659} C_VEL
LIN {X 0,Y 290.552,Z 551.39,A -85,B 0,C 180,E1 -19850.07,E2 -19850.07} C_VEL
LIN {X 0,Y 279.502,Z 602.269,A -85,B 0,C 180,E1 -19852.428,E2 -19852.428} C_VEL
LIN {X 0,Y 275.668,Z 615.402,A -85,B 0,C 180,E1 -19853.193,E2 -19853.193} C_VEL
LIN {X 0,Y 270.902,Z 629.049,A -85,B 0,C 180,E1 -19854.287,E2 -19854.287} C_VEL
LIN {X 0,Y 265.788,Z 641.252,A -85,B 0,C 180,E1 -19855.584,E2 -19855.584} C_VEL
LIN {X 0,Y 260.024,Z 653.375,A -85,B 0,C 180,E1 -19857.278,E2 -19857.278} C_VEL
LIN {X 0,Y 254.196,Z 664.051,A -85,B 0,C 180,E1 -19859.237,E2 -19859.237} C_VEL
LIN {X 0,Y 249,Z 672.881,A -85,B 0,C 180,E1 -19861.326,E2 -19861.326} C_VEL
LIN {X 0,Y 244.163,Z 680.259,A -85,B 0,C 180,E1 -19863.565,E2 -19863.565} C_VEL
LIN {X 0,Y 239.996,Z 686.138,A -85,B 0,C 180,E1 -19865.797,E2 -19865.797} C_VEL
LIN {X 0,Y 236.338,Z 690.964,A -85,B 0,C 180,E1 -19868.179,E2 -19868.179} C_VEL
LIN {X 0,Y 233.114,Z 694.815,A -85,B 0,C 180,E1 -19870.632,E2 -19870.632} C_VEL
LIN {X 0,Y 229.925,Z 698.434,A -85,B 0,C 180,E1 -19874.032,E2 -19874.032} C_VEL
LIN {X 0,Y 227.64,Z 700.432,A -85,B 0,C 180,E1 -19877.519,E2 -19877.519} C_VEL
LIN {X 0,Y 226.318,Z 700.901,A -85,B 0,C 180,E1 -19881.068,E2 -19881.068} C_VEL
LIN {X 0,Y 225.816,Z 700.067,A -85,B 0,C 180,E1 -19884.419,E2 -19884.419} C_VEL
LIN {X 0,Y 225.702,Z 701.217,A -85,B 0,C 180,E1 -19886.429,E2 -19886.429} C_VEL
LIN {X 0,Y 225.733,Z 701.833,A -85,B 0,C 180,E1 -19888.216,E2 -19888.216} C_VEL
LIN {X 0,Y 225.774,Z 702.05,A -85,B 0,C 180,E1 -19890,E2 -19890} C_VEL
LIN {X 0,Y 225.701,Z 701.821,A -85,B 0,C 180,E1 -19891.784,E2 -19891.784} C_VEL
LIN {X 0,Y 225.679,Z 700.555,A -85,B 0,C 180,E1 -19894.771,E2 -19894.771} C_VEL
LIN {X 0,Y 225.842,Z 698.742,A -85,B 0,C 180,E1 -19897.151,E2 -19897.151} C_VEL
LIN {X 0,Y 226.35,Z 695.757,A -85,B 0,C 180,E1 -19899.833,E2 -19899.833} C_VEL
LIN {X 0,Y 227.193,Z 691.709,A -85,B 0,C 180,E1 -19902.506,E2 -19902.506} C_VEL
LIN {X 0,Y 228.763,Z 685.475,A -85,B 0,C 180,E1 -19905.594,E2 -19905.594} C_VEL
LIN {X 0,Y 230.561,Z 678.679,A -85,B 0,C 180,E1 -19908.207,E2 -19908.207} C_VEL
LIN {X 0,Y 232.804,Z 670.289,A -85,B 0,C 180,E1 -19910.789,E2 -19910.789} C_VEL
LIN {X 0,Y 236.462,Z 664.805,A -85,B 0,C 180,E1 -19913.656,E2 -19913.656} C_VEL
LIN {X 0,Y 241.088,Z 657.878,A -85,B 0,C 180,E1 -19916.395,E2 -19916.395} C_VEL
LIN {X 0,Y 245.712,Z 650.683,A -85,B 0,C 180,E1 -19918.626,E2 -19918.626} C_VEL
LIN {X 0,Y 250.935,Z 642.107,A -85,B 0,C 180,E1 -19920.739,E2 -19920.739} C_VEL
LIN {X 0,Y 256.708,Z 631.871,A -85,B 0,C 180,E1 -19922.732,E2 -19922.732} C_VEL
LIN {X 0,Y 262.652,Z 620.469,A -85,B 0,C 180,E1 -19924.421,E2 -19924.421} C_VEL
LIN {X 0,Y 267.877,Z 609.178,A -85,B 0,C 180,E1 -19925.761,E2 -19925.761} C_VEL
LIN {X 0,Y 273.452,Z 595.327,A -85,B 0,C 180,E1 -19927.021,E2 -19927.021} C_VEL
LIN {X 0,Y 278.253,Z 581.249,A -85,B 0,C 180,E1 -19927.964,E2 -19927.964} C_VEL
LIN {X 0,Y 282.355,Z 565.677,A -85,B 0,C 180,E1 -19928.806,E2 -19928.806} C_VEL
LIN {X 0,Y 286.332,Z 546.434,A -85,B 0,C 180,E1 -19929.713,E2 -19929.713} C_VEL
LIN {X 0,Y 287.704,Z 537.217,A -85,B 0,C 180,E1 -19930.58,E2 -19930.58} C_VEL
LIN {X 0,Y 288.335,Z 532.244,A -85,B 0,C 180,E1 -19931.2,E2 -19931.2} C_VEL
LIN {X 0,Y 287.974,Z 528.045,A -85,B 0,C 180,E1 -19932.859,E2 -19932.859} C_VEL
LIN {X 0,Y 287.824,Z 524.6,A -85,B 0,C 180,E1 -19935.273,E2 -19935.273} C_VEL
LIN {X 0,Y 288.142,Z 523.374,A -85,B 0,C 180,E1 -19937.031,E2 -19937.031} C_VEL
LIN {X 0,Y 289.349,Z 523.142,A -85,B 0,C 180,E1 -19939.555,E2 -19939.555} C_VEL
LIN {X 0,Y 290.322,Z 524.184,A -85,B 0,C 180,E1 -19940.952,E2 -19940.952} C_VEL
LIN {X 0,Y 284.642,Z 550.853,A -85,B 0,C 180,E1 -19942.275,E2 -19942.275} C_VEL
LIN {X 0,Y 281.877,Z 562.399,A -85,B 0,C 180,E1 -19943.022,E2 -19943.022} C_VEL
LIN {X 0,Y 278.283,Z 574.496,A -85,B 0,C 180,E1 -19944.043,E2 -19944.043} C_VEL
LIN {X 0,Y 273.778,Z 586.901,A -85,B 0,C 180,E1 -19945.392,E2 -19945.392} C_VEL
LIN {X 0,Y 268.905,Z 598.103,A -85,B 0,C 180,E1 -19946.936,E2 -19946.936} C_VEL
LIN {X 0,Y 263.784,Z 608.265,A -85,B 0,C 180,E1 -19948.699,E2 -19948.699} C_VEL
LIN {X 0,Y 258.506,Z 617.31,A -85,B 0,C 180,E1 -19950.701,E2 -19950.701} C_VEL
LIN {X 0,Y 253.304,Z 625.26,A -85,B 0,C 180,E1 -19952.978,E2 -19952.978} C_VEL
LIN {X 0,Y 249.148,Z 630.778,A -85,B 0,C 180,E1 -19954.968,E2 -19954.968} C_VEL
LIN {X 0,Y 245.06,Z 635.646,A -85,B 0,C 180,E1 -19957.222,E2 -19957.222} C_VEL
LIN {X 0,Y 241.3,Z 639.453,A -85,B 0,C 180,E1 -19959.543,E2 -19959.543} C_VEL
LIN {X 0,Y 236.863,Z 642.967,A -85,B 0,C 180,E1 -19962.74,E2 -19962.74} C_VEL
LIN {X 0,Y 234.947,Z 644.128,A -85,B 0,C 180,E1 -19964.382,E2 -19964.382} C_VEL
LIN {X 0,Y 233.194,Z 644.882,A -85,B 0,C 180,E1 -19966.048,E2 -19966.048} C_VEL
LIN {X 0,Y 230.444,Z 645.113,A -85,B 0,C 180,E1 -19969.456,E2 -19969.456} C_VEL
LIN {X 0,Y 228.512,Z 643.794,A -85,B 0,C 180,E1 -19972.934,E2 -19972.934} C_VEL
LIN {X 0,Y 227.756,Z 642.509,A -85,B 0,C 180,E1 -19974.688,E2 -19974.688} C_VEL
LIN {X 0,Y 226.873,Z 639.838,A -85,B 0,C 180,E1 -19977.337,E2 -19977.337} C_VEL
LIN {X 0,Y 226.445,Z 636.149,A -85,B 0,C 180,E1 -19980,E2 -19980} C_VEL
LIN {X 0,Y 226.452,Z 631.394,A -85,B 0,C 180,E1 -19982.668,E2 -19982.668} C_VEL
LIN {X 0,Y 226.771,Z 625.456,A -85,B 0,C 180,E1 -19985.335,E2 -19985.335} C_VEL
LIN {X 0,Y 226.994,Z 618.092,A -85,B 0,C 180,E1 -19988.008,E2 -19988.008} C_VEL
LIN {X 0,Y 227.599,Z 609.009,A -85,B 0,C 180,E1 -19990.677,E2 -19990.677} C_VEL
LIN {X 0,Y 228.42,Z 598.751,A -85,B 0,C 180,E1 -19993.116,E2 -19993.116} C_VEL
LIN {X 0,Y 229.416,Z 587.367,A -85,B 0,C 180,E1 -19995.321,E2 -19995.321} C_VEL
LIN {X 0,Y 230.398,Z 574.587,A -85,B 0,C 180,E1 -19997.302,E2 -19997.302} C_VEL
LIN {X 0,Y 231.351,Z 562.108,A -85,B 0,C 180,E1 -19998.831,E2 -19998.831} C_VEL
LIN {X 0,Y 232.054,Z 549.126,A -85,B 0,C 180,E1 -20000.066,E2 -20000.066} C_VEL
LIN {X 0,Y 232.754,Z 535.596,A -85,B 0,C 180,E1 -20001.007,E2 -20001.007} C_VEL
LIN {X 0,Y 235.33,Z 470.636,A -85,B 0,C 180,E1 -20004.269,E2 -20004.269} C_VEL
LIN {X 0,Y 228.699,Z 447.917,A -85,B 0,C 180,E1 -20005.74,E2 -20005.74} C_VEL
LIN {X 0,Y 227.975,Z 445.087,A -85,B 0,C 180,E1 -20005.967,E2 -20005.967} C_VEL
LIN {X 0,Y 227.899,Z 445.097,A -85,B 0,C 180,E1 -20010.291,E2 -20010.291} C_VEL
LIN {X 0,Y 227.879,Z 445.063,A -85,B 0,C 180,E1 -20013.72,E2 -20013.72} C_VEL
LIN {X 0,Y 227.846,Z 445.102,A -85,B 0,C 180,E1 -20018.091,E2 -20018.091} C_VEL
LIN {X 0,Y 227.812,Z 445.107,A -85,B 0,C 180,E1 -20022.743,E2 -20022.743} C_VEL
LIN {X 0,Y 227.846,Z 445.103,A -85,B 0,C 180,E1 -20024.51,E2 -20024.51} C_VEL
LIN {X 0,Y 231.721,Z 455.888,A -85,B 0,C 180,E1 -20028.582,E2 -20028.582} C_VEL
LIN {X 0,Y 234.931,Z 465.916,A -85,B 0,C 180,E1 -20032,E2 -20032} C_VEL
LIN {X 0,Y 237.45,Z 475.372,A -85,B 0,C 180,E1 -20034.898,E2 -20034.898} C_VEL
LIN {X 0,Y 244.44,Z 490.819,A -85,B 0,C 180,E1 -20036.582,E2 -20036.582} C_VEL
LIN {X 0,Y 245.783,Z 494.893,A -85,B 0,C 180,E1 -20036.929,E2 -20036.929} C_VEL
LIN {X 0,Y 248.95,Z 515.144,A -85,B 0,C 180,E1 -20038.084,E2 -20038.084} C_VEL
LIN {X 0,Y 246.291,Z 584.473,A -85,B 0,C 180,E1 -20040.042,E2 -20040.042} C_VEL
LIN {X 0,Y 245.246,Z 598.013,A -85,B 0,C 180,E1 -20040.669,E2 -20040.669} C_VEL
LIN {X 0,Y 243.908,Z 609.633,A -85,B 0,C 180,E1 -20041.495,E2 -20041.495} C_VEL
LIN {X 0,Y 242.292,Z 620.756,A -85,B 0,C 180,E1 -20042.582,E2 -20042.582} C_VEL
LIN {X 0,Y 240.27,Z 631.729,A -85,B 0,C 180,E1 -20043.975,E2 -20043.975} C_VEL
LIN {X 0,Y 237.865,Z 642.92,A -85,B 0,C 180,E1 -20045.798,E2 -20045.798} C_VEL
LIN {X 0,Y 235.624,Z 652.542,A -85,B 0,C 180,E1 -20047.798,E2 -20047.798} C_VEL
LIN {X 0,Y 233.69,Z 660.217,A -85,B 0,C 180,E1 -20049.766,E2 -20049.766} C_VEL
LIN {X 0,Y 231.319,Z 668.264,A -85,B 0,C 180,E1 -20052.313,E2 -20052.313} C_VEL
LIN {X 0,Y 229.551,Z 674.728,A -85,B 0,C 180,E1 -20054.916,E2 -20054.916} C_VEL
LIN {X 0,Y 228.08,Z 679.868,A -85,B 0,C 180,E1 -20057.544,E2 -20057.544} C_VEL
LIN {X 0,Y 227.021,Z 683.844,A -85,B 0,C 180,E1 -20060.197,E2 -20060.197} C_VEL
LIN {X 0,Y 226.324,Z 686.772,A -85,B 0,C 180,E1 -20062.865,E2 -20062.865} C_VEL
LIN {X 0,Y 226.011,Z 688.189,A -85,B 0,C 180,E1 -20064.647,E2 -20064.647} C_VEL
LIN {X 0,Y 225.745,Z 689.793,A -85,B 0,C 180,E1 -20068.216,E2 -20068.216} C_VEL
LIN {X 0,Y 225.719,Z 690.024,A -85,B 0,C 180,E1 -20070,E2 -20070} C_VEL
LIN {X 0,Y 225.745,Z 689.828,A -85,B 0,C 180,E1 -20071.784,E2 -20071.784} C_VEL
LIN {X 0,Y 226.011,Z 688.269,A -85,B 0,C 180,E1 -20075.353,E2 -20075.353} C_VEL
LIN {X 0,Y 226.322,Z 686.897,A -85,B 0,C 180,E1 -20077.135,E2 -20077.135} C_VEL
LIN {X 0,Y 227.004,Z 684.016,A -85,B 0,C 180,E1 -20079.804,E2 -20079.804} C_VEL
LIN {X 0,Y 228.033,Z 680.098,A -85,B 0,C 180,E1 -20082.459,E2 -20082.459} C_VEL
LIN {X 0,Y 229.514,Z 675.016,A -85,B 0,C 180,E1 -20085.087,E2 -20085.087} C_VEL
LIN {X 0,Y 231.306,Z 668.609,A -85,B 0,C 180,E1 -20087.688,E2 -20087.688} C_VEL
LIN {X 0,Y 233.642,Z 660.641,A -85,B 0,C 180,E1 -20090.238,E2 -20090.238} C_VEL
LIN {X 0,Y 235.95,Z 651.48,A -85,B 0,C 180,E1 -20092.576,E2 -20092.576} C_VEL
LIN {X 0,Y 238.295,Z 641.311,A -85,B 0,C 180,E1 -20094.619,E2 -20094.619} C_VEL
LIN {X 0,Y 240.478,Z 631.152,A -85,B 0,C 180,E1 -20096.234,E2 -20096.234} C_VEL
LIN {X 0,Y 242.473,Z 620.014,A -85,B 0,C 180,E1 -20097.63,E2 -20097.63} C_VEL
LIN {X 0,Y 244.344,Z 607.371,A -85,B 0,C 180,E1 -20098.802,E2 -20098.802} C_VEL
LIN {X 0,Y 245.619,Z 594.896,A -85,B 0,C 180,E1 -20099.635,E2 -20099.635} C_VEL
LIN {X 0,Y 246.511,Z 581.954,A -85,B 0,C 180,E1 -20100.165,E2 -20100.165} C_VEL
LIN {X 0,Y 248.988,Z 514.874,A -85,B 0,C 180,E1 -20102.057,E2 -20102.057} C_VEL
LIN {X 0,Y 245.524,Z 493.36,A -85,B 0,C 180,E1 -20103.304,E2 -20103.304} C_VEL
LIN {X 0,Y 239.147,Z 478.875,A -85,B 0,C 180,E1 -20104.834,E2 -20104.834} C_VEL
LIN {X 0,Y 237.417,Z 475.189,A -85,B 0,C 180,E1 -20105.277,E2 -20105.277} C_VEL
LIN {X 0,Y 234.369,Z 464.007,A -85,B 0,C 180,E1 -20108.77,E2 -20108.77} C_VEL
LIN {X 0,Y 231.439,Z 455,A -85,B 0,C 180,E1 -20111.918,E2 -20111.918} C_VEL
LIN {X 0,Y 228.988,Z 448.154,A -85,B 0,C 180,E1 -20114.473,E2 -20114.473} C_VEL
LIN {X 0,Y 227.858,Z 445.107,A -85,B 0,C 180,E1 -20115.739,E2 -20115.739} C_VEL
LIN {X 0,Y 227.854,Z 445.105,A -85,B 0,C 180,E1 -20120.454,E2 -20120.454} C_VEL
LIN {X 0,Y 227.977,Z 445.193,A -85,B 0,C 180,E1 -20125.294,E2 -20125.294} C_VEL
LIN {X 0,Y 231.347,Z 461.259,A -85,B 0,C 180,E1 -20129.665,E2 -20129.665} C_VEL
LIN {X 0,Y 233.202,Z 470.725,A -85,B 0,C 180,E1 -20132.152,E2 -20132.152} C_VEL
LIN {X 0,Y 232.773,Z 475.866,A -85,B 0,C 180,E1 -20133.417,E2 -20133.417} C_VEL
LIN {X 0,Y 234.383,Z 496.925,A -85,B 0,C 180,E1 -20134.58,E2 -20134.58} C_VEL
LIN {X 0,Y 235.771,Z 509.727,A -85,B 0,C 180,E1 -20135.287,E2 -20135.287} C_VEL
LIN {X 0,Y 233.293,Z 564.571,A -85,B 0,C 180,E1 -20138.011,E2 -20138.011} C_VEL
LIN {X 0,Y 232.404,Z 570.307,A -85,B 0,C 180,E1 -20138.283,E2 -20138.283} C_VEL
LIN {X 0,Y 225.897,Z 588.691,A -85,B 0,C 180,E1 -20139.204,E2 -20139.204} C_VEL
LIN {X 0,Y 224.797,Z 594.299,A -85,B 0,C 180,E1 -20139.603,E2 -20139.603} C_VEL
LIN {X 0,Y 223.958,Z 608.384,A -85,B 0,C 180,E1 -20140.874,E2 -20140.874} C_VEL
LIN {X 0,Y 222.855,Z 622.309,A -85,B 0,C 180,E1 -20142.567,E2 -20142.567} C_VEL
LIN {X 0,Y 221.901,Z 633.985,A -85,B 0,C 180,E1 -20144.383,E2 -20144.383} C_VEL
LIN {X 0,Y 220.943,Z 644.702,A -85,B 0,C 180,E1 -20146.432,E2 -20146.432} C_VEL
LIN {X 0,Y 220.054,Z 655.332,A -85,B 0,C 180,E1 -20148.952,E2 -20148.952} C_VEL
LIN {X 0,Y 219.506,Z 663.277,A -85,B 0,C 180,E1 -20151.252,E2 -20151.252} C_VEL
LIN {X 0,Y 219.008,Z 671.353,A -85,B 0,C 180,E1 -20154.154,E2 -20154.154} C_VEL
LIN {X 0,Y 218.828,Z 678.169,A -85,B 0,C 180,E1 -20157.239,E2 -20157.239} C_VEL
LIN {X 0,Y 218.714,Z 682.884,A -85,B 0,C 180,E1 -20160,E2 -20160} C_VEL
LIN {X 0,Y 218.789,Z 686.461,A -85,B 0,C 180,E1 -20162.762,E2 -20162.762} C_VEL
LIN {X 0,Y 219.294,Z 689.704,A -85,B 0,C 180,E1 -20166.535,E2 -20166.535} C_VEL
LIN {X 0,Y 220.155,Z 690.983,A -85,B 0,C 180,E1 -20169.184,E2 -20169.184} C_VEL
LIN {X 0,Y 222.044,Z 691.413,A -85,B 0,C 180,E1 -20172.801,E2 -20172.801} C_VEL
LIN {X 0,Y 224.844,Z 690.231,A -85,B 0,C 180,E1 -20176.339,E2 -20176.339} C_VEL
LIN {X 0,Y 226.484,Z 689.094,A -85,B 0,C 180,E1 -20178.078,E2 -20178.078} C_VEL
LIN {X 0,Y 229.732,Z 686.576,A -85,B 0,C 180,E1 -20180.598,E2 -20180.598} C_VEL
LIN {X 0,Y 233.324,Z 683.116,A -85,B 0,C 180,E1 -20183.053,E2 -20183.053} C_VEL
LIN {X 0,Y 237.408,Z 678.691,A -85,B 0,C 180,E1 -20185.42,E2 -20185.42} C_VEL
LIN {X 0,Y 242.838,Z 672.064,A -85,B 0,C 180,E1 -20188.053,E2 -20188.053} C_VEL
LIN {X 0,Y 247.966,Z 665.041,A -85,B 0,C 180,E1 -20190.204,E2 -20190.204} C_VEL
LIN {X 0,Y 253.491,Z 656.529,A -85,B 0,C 180,E1 -20192.256,E2 -20192.256} C_VEL
LIN {X 0,Y 259.428,Z 646.187,A -85,B 0,C 180,E1 -20194.203,E2 -20194.203} C_VEL
LIN {X 0,Y 265.281,Z 634.554,A -85,B 0,C 180,E1 -20195.884,E2 -20195.884} C_VEL
LIN {X 0,Y 270.301,Z 622.903,A -85,B 0,C 180,E1 -20197.194,E2 -20197.194} C_VEL
LIN {X 0,Y 275.621,Z 608.078,A -85,B 0,C 180,E1 -20198.428,E2 -20198.428} C_VEL
LIN {X 0,Y 279.649,Z 593.845,A -85,B 0,C 180,E1 -20199.272,E2 -20199.272} C_VEL
LIN {X 0,Y 290.899,Z 544.366,A -85,B 0,C 180,E1 -20201.5,E2 -20201.5} C_VEL
LIN {X 0,Y 290.681,Z 542.433,A -85,B 0,C 180,E1 -20202.695,E2 -20202.695} C_VEL
LIN {X 0,Y 290.594,Z 540.84,A -85,B 0,C 180,E1 -20204.316,E2 -20204.316} C_VEL
LIN {X 0,Y 290.881,Z 540.535,A -85,B 0,C 180,E1 -20206.455,E2 -20206.455} C_VEL
LIN {X 0,Y 291.366,Z 540.924,A -85,B 0,C 180,E1 -20207.763,E2 -20207.763} C_VEL
LIN {X 0,Y 289.877,Z 548.325,A -85,B 0,C 180,E1 -20208.455,E2 -20208.455} C_VEL
LIN {X 0,Y 288.608,Z 553.963,A -85,B 0,C 180,E1 -20208.778,E2 -20208.778} C_VEL
LIN {X 0,Y 277.647,Z 601.589,A -85,B 0,C 180,E1 -20210.975,E2 -20210.975} C_VEL
LIN {X 0,Y 273.016,Z 616.614,A -85,B 0,C 180,E1 -20211.843,E2 -20211.843} C_VEL
LIN {X 0,Y 268.007,Z 629.784,A -85,B 0,C 180,E1 -20212.905,E2 -20212.905} C_VEL
LIN {X 0,Y 262.079,Z 642.852,A -85,B 0,C 180,E1 -20214.32,E2 -20214.32} C_VEL
LIN {X 0,Y 256.572,Z 653.515,A -85,B 0,C 180,E1 -20215.838,E2 -20215.838} C_VEL
LIN {X 0,Y 250.397,Z 664.08,A -85,B 0,C 180,E1 -20217.772,E2 -20217.772} C_VEL
LIN {X 0,Y 244.783,Z 672.745,A -85,B 0,C 180,E1 -20219.838,E2 -20219.838} C_VEL
LIN {X 0,Y 238.89,Z 681.023,A -85,B 0,C 180,E1 -20222.396,E2 -20222.396} C_VEL
LIN {X 0,Y 233.666,Z 687.577,A -85,B 0,C 180,E1 -20225.097,E2 -20225.097} C_VEL
LIN {X 0,Y 229.851,Z 692.062,A -85,B 0,C 180,E1 -20227.53,E2 -20227.53} C_VEL
LIN {X 0,Y 226.489,Z 695.54,A -85,B 0,C 180,E1 -20230.042,E2 -20230.042} C_VEL
LIN {X 0,Y 223.097,Z 698.738,A -85,B 0,C 180,E1 -20233.53,E2 -20233.53} C_VEL
LIN {X 0,Y 220.701,Z 700.409,A -85,B 0,C 180,E1 -20237.12,E2 -20237.12} C_VEL
LIN {X 0,Y 219.304,Z 700.49,A -85,B 0,C 180,E1 -20240.779,E2 -20240.779} C_VEL
LIN {X 0,Y 218.803,Z 699.532,A -85,B 0,C 180,E1 -20243.777,E2 -20243.777} C_VEL
LIN {X 0,Y 218.617,Z 701.028,A -85,B 0,C 180,E1 -20246.314,E2 -20246.314} C_VEL
LIN {X 0,Y 218.629,Z 701.644,A -85,B 0,C 180,E1 -20248.158,E2 -20248.158} C_VEL
LIN {X 0,Y 218.686,Z 701.862,A -85,B 0,C 180,E1 -20250,E2 -20250} C_VEL
LIN {X 0,Y 218.597,Z 701.632,A -85,B 0,C 180,E1 -20251.842,E2 -20251.842} C_VEL
LIN {X 0,Y 218.569,Z 700.572,A -85,B 0,C 180,E1 -20254.588,E2 -20254.588} C_VEL
LIN {X 0,Y 218.793,Z 698.553,A -85,B 0,C 180,E1 -20257.382,E2 -20257.382} C_VEL
LIN {X 0,Y 219.33,Z 695.567,A -85,B 0,C 180,E1 -20260.151,E2 -20260.151} C_VEL
LIN {X 0,Y 220.21,Z 691.518,A -85,B 0,C 180,E1 -20262.909,E2 -20262.909} C_VEL
LIN {X 0,Y 221.895,Z 685.286,A -85,B 0,C 180,E1 -20266.089,E2 -20266.089} C_VEL
LIN {X 0,Y 223.813,Z 678.491,A -85,B 0,C 180,E1 -20268.776,E2 -20268.776} C_VEL
LIN {X 0,Y 225.984,Z 670.753,A -85,B 0,C 180,E1 -20271.268,E2 -20271.268} C_VEL
LIN {X 0,Y 230.007,Z 665.43,A -85,B 0,C 180,E1 -20274.362,E2 -20274.362} C_VEL
LIN {X 0,Y 234.842,Z 658.995,A -85,B 0,C 180,E1 -20277.154,E2 -20277.154} C_VEL
LIN {X 0,Y 239.639,Z 652.283,A -85,B 0,C 180,E1 -20279.422,E2 -20279.422} C_VEL
LIN {X 0,Y 245.034,Z 644.299,A -85,B 0,C 180,E1 -20281.563,E2 -20281.563} C_VEL
LIN {X 0,Y 250.971,Z 634.79,A -85,B 0,C 180,E1 -20283.578,E2 -20283.578} C_VEL
LIN {X 0,Y 257.049,Z 624.302,A -85,B 0,C 180,E1 -20285.281,E2 -20285.281} C_VEL
LIN {X 0,Y 263.174,Z 612.418,A -85,B 0,C 180,E1 -20286.817,E2 -20286.817} C_VEL
LIN {X 0,Y 269.491,Z 598.382,A -85,B 0,C 180,E1 -20288.176,E2 -20288.176} C_VEL
LIN {X 0,Y 274.399,Z 585.596,A -85,B 0,C 180,E1 -20289.102,E2 -20289.102} C_VEL
LIN {X 0,Y 279.052,Z 570.659,A -85,B 0,C 180,E1 -20289.961,E2 -20289.961} C_VEL
LIN {X 0,Y 284.279,Z 547.834,A -85,B 0,C 180,E1 -20291.06,E2 -20291.06} C_VEL
LIN {X 0,Y 285.858,Z 538.614,A -85,B 0,C 180,E1 -20291.975,E2 -20291.975} C_VEL
LIN {X 0,Y 286.037,Z 537.317,A -85,B 0,C 180,E1 -20292.177,E2 -20292.177} C_VEL
LIN {X 0,Y 285.956,Z 534.364,A -85,B 0,C 180,E1 -20293.387,E2 -20293.387} C_VEL
LIN {X 0,Y 285.997,Z 531.218,A -85,B 0,C 180,E1 -20295.644,E2 -20295.644} C_VEL
LIN {X 0,Y 286.267,Z 530.313,A -85,B 0,C 180,E1 -20296.911,E2 -20296.911} C_VEL
LIN {X 0,Y 287.357,Z 529.961,A -85,B 0,C 180,E1 -20299.304,E2 -20299.304} C_VEL
LIN {X 0,Y 287.647,Z 530.35,A -85,B 0,C 180,E1 -20299.851,E2 -20299.851} C_VEL
LIN {X 0,Y 282.637,Z 552.462,A -85,B 0,C 180,E1 -20300.942,E2 -20300.942} C_VEL
LIN {X 0,Y 279.987,Z 562.817,A -85,B 0,C 180,E1 -20301.592,E2 -20301.592} C_VEL
LIN {X 0,Y 275.671,Z 576.383,A -85,B 0,C 180,E1 -20302.736,E2 -20302.736} C_VEL
LIN {X 0,Y 270.651,Z 589.125,A -85,B 0,C 180,E1 -20304.135,E2 -20304.135} C_VEL
LIN {X 0,Y 265.008,Z 600.981,A -85,B 0,C 180,E1 -20305.813,E2 -20305.813} C_VEL
LIN {X 0,Y 259.367,Z 611.094,A -85,B 0,C 180,E1 -20307.645,E2 -20307.645} C_VEL
LIN {X 0,Y 253.821,Z 619.775,A -85,B 0,C 180,E1 -20309.647,E2 -20309.647} C_VEL
LIN {X 0,Y 248.707,Z 626.85,A -85,B 0,C 180,E1 -20311.75,E2 -20311.75} C_VEL
LIN {X 0,Y 243.131,Z 633.488,A -85,B 0,C 180,E1 -20314.304,E2 -20314.304} C_VEL
LIN {X 0,Y 238.844,Z 637.942,A -85,B 0,C 180,E1 -20316.594,E2 -20316.594} C_VEL
LIN {X 0,Y 234.915,Z 641.402,A -85,B 0,C 180,E1 -20318.961,E2 -20318.961} C_VEL
LIN {X 0,Y 232.513,Z 643.19,A -85,B 0,C 180,E1 -20320.58,E2 -20320.58} C_VEL
LIN {X 0,Y 230.262,Z 644.552,A -85,B 0,C 180,E1 -20322.229,E2 -20322.229} C_VEL
LIN {X 0,Y 226.413,Z 646.025,A -85,B 0,C 180,E1 -20325.622,E2 -20325.622} C_VEL
LIN {X 0,Y 224.839,Z 646.185,A -85,B 0,C 180,E1 -20327.361,E2 -20327.361} C_VEL
LIN {X 0,Y 223.522,Z 645.944,A -85,B 0,C 180,E1 -20329.126,E2 -20329.126} C_VEL
LIN {X 0,Y 221.494,Z 644.228,A -85,B 0,C 180,E1 -20332.708,E2 -20332.708} C_VEL
LIN {X 0,Y 220.033,Z 640.946,A -85,B 0,C 180,E1 -20336.337,E2 -20336.337} C_VEL
LIN {X 0,Y 219.45,Z 637.349,A -85,B 0,C 180,E1 -20339.083,E2 -20339.083} C_VEL
LIN {X 0,Y 219.327,Z 632.7,A -85,B 0,C 180,E1 -20341.836,E2 -20341.836} C_VEL
LIN {X 0,Y 219.665,Z 625.742,A -85,B 0,C 180,E1 -20345.048,E2 -20345.048} C_VEL
LIN {X 0,Y 219.825,Z 618.731,A -85,B 0,C 180,E1 -20347.649,E2 -20347.649} C_VEL
LIN {X 0,Y 220.342,Z 610.761,A -85,B 0,C 180,E1 -20350.104,E2 -20350.104} C_VEL
LIN {X 0,Y 221.137,Z 600.835,A -85,B 0,C 180,E1 -20352.621,E2 -20352.621} C_VEL
LIN {X 0,Y 222.067,Z 589.718,A -85,B 0,C 180,E1 -20354.901,E2 -20354.901} C_VEL
LIN {X 0,Y 222.963,Z 578.892,A -85,B 0,C 180,E1 -20356.716,E2 -20356.716} C_VEL
LIN {X 0,Y 224.031,Z 565.433,A -85,B 0,C 180,E1 -20358.52,E2 -20358.52} C_VEL
LIN {X 0,Y 224.76,Z 552.281,A -85,B 0,C 180,E1 -20359.88,E2 -20359.88} C_VEL
LIN {X 0,Y 225.585,Z 538.039,A -85,B 0,C 180,E1 -20360.968,E2 -20360.968} C_VEL
LIN {X 0,Y 228.239,Z 471.763,A -85,B 0,C 180,E1 -20364.493,E2 -20364.493} C_VEL
LIN {X 0,Y 221.058,Z 446.661,A -85,B 0,C 180,E1 -20366.135,E2 -20366.135} C_VEL
LIN {X 0,Y 220.929,Z 445.964,A -85,B 0,C 180,E1 -20366.183,E2 -20366.183} C_VEL
LIN {X 0,Y 220.84,Z 445.971,A -85,B 0,C 180,E1 -20370.768,E2 -20370.768} C_VEL
LIN {X 0,Y 220.803,Z 445.95,A -85,B 0,C 180,E1 -20374.955,E2 -20374.955} C_VEL
LIN {X 0,Y 220.808,Z 445.959,A -85,B 0,C 180,E1 -20379.537,E2 -20379.537} C_VEL
LIN {X 0,Y 220.786,Z 446.017,A -85,B 0,C 180,E1 -20382.985,E2 -20382.985} C_VEL
LIN {X 0,Y 224.796,Z 456.769,A -85,B 0,C 180,E1 -20387.281,E2 -20387.281} C_VEL
LIN {X 0,Y 228.137,Z 466.922,A -85,B 0,C 180,E1 -20390.938,E2 -20390.938} C_VEL
LIN {X 0,Y 230.592,Z 475.723,A -85,B 0,C 180,E1 -20393.7,E2 -20393.7} C_VEL
LIN {X 0,Y 237.645,Z 490.899,A -85,B 0,C 180,E1 -20395.493,E2 -20395.493} C_VEL
LIN {X 0,Y 239.973,Z 496.793,A -85,B 0,C 180,E1 -20396.085,E2 -20396.085} C_VEL
LIN {X 0,Y 242.918,Z 516.127,A -85,B 0,C 180,E1 -20397.224,E2 -20397.224} C_VEL
LIN {X 0,Y 240.108,Z 585.925,A -85,B 0,C 180,E1 -20399.249,E2 -20399.249} C_VEL
LIN {X 0,Y 239.011,Z 599.017,A -85,B 0,C 180,E1 -20399.886,E2 -20399.886} C_VEL
LIN {X 0,Y 237.566,Z 610.938,A -85,B 0,C 180,E1 -20400.782,E2 -20400.782} C_VEL
LIN {X 0,Y 235.686,Z 622.634,A -85,B 0,C 180,E1 -20401.988,E2 -20401.988} C_VEL
LIN {X 0,Y 233.351,Z 634.667,A -85,B 0,C 180,E1 -20403.625,E2 -20403.625} C_VEL
LIN {X 0,Y 230.893,Z 645.254,A -85,B 0,C 180,E1 -20405.498,E2 -20405.498} C_VEL
LIN {X 0,Y 228.493,Z 655.053,A -85,B 0,C 180,E1 -20407.704,E2 -20407.704} C_VEL
LIN {X 0,Y 226.173,Z 663.307,A -85,B 0,C 180,E1 -20410.013,E2 -20410.013} C_VEL
LIN {X 0,Y 223.891,Z 670.772,A -85,B 0,C 180,E1 -20412.65,E2 -20412.65} C_VEL
LIN {X 0,Y 222.132,Z 676.756,A -85,B 0,C 180,E1 -20415.338,E2 -20415.338} C_VEL
LIN {X 0,Y 220.709,Z 681.487,A -85,B 0,C 180,E1 -20418.055,E2 -20418.055} C_VEL
LIN {X 0,Y 219.746,Z 685.101,A -85,B 0,C 180,E1 -20420.798,E2 -20420.798} C_VEL
LIN {X 0,Y 219.008,Z 688.168,A -85,B 0,C 180,E1 -20424.154,E2 -20424.154} C_VEL
LIN {X 0,Y 218.74,Z 689.371,A -85,B 0,C 180,E1 -20426.316,E2 -20426.316} C_VEL
LIN {X 0,Y 218.665,Z 689.982,A -85,B 0,C 180,E1 -20428.158,E2 -20428.158} C_VEL
LIN {X 0,Y 218.635,Z 690.213,A -85,B 0,C 180,E1 -20430,E2 -20430} C_VEL
LIN {X 0,Y 218.664,Z 690.016,A -85,B 0,C 180,E1 -20431.842,E2 -20431.842} C_VEL
LIN {X 0,Y 218.955,Z 688.457,A -85,B 0,C 180,E1 -20435.526,E2 -20435.526} C_VEL
LIN {X 0,Y 219.273,Z 687.085,A -85,B 0,C 180,E1 -20437.366,E2 -20437.366} C_VEL
LIN {X 0,Y 219.99,Z 684.204,A -85,B 0,C 180,E1 -20440.12,E2 -20440.12} C_VEL
LIN {X 0,Y 221.09,Z 680.285,A -85,B 0,C 180,E1 -20442.857,E2 -20442.857} C_VEL
LIN {X 0,Y 222.666,Z 675.201,A -85,B 0,C 180,E1 -20445.562,E2 -20445.562} C_VEL
LIN {X 0,Y 224.562,Z 668.793,A -85,B 0,C 180,E1 -20448.238,E2 -20448.238} C_VEL
LIN {X 0,Y 226.996,Z 660.823,A -85,B 0,C 180,E1 -20450.858,E2 -20450.858} C_VEL
LIN {X 0,Y 229.254,Z 652.26,A -85,B 0,C 180,E1 -20453.12,E2 -20453.12} C_VEL
LIN {X 0,Y 231.57,Z 642.628,A -85,B 0,C 180,E1 -20455.144,E2 -20455.144} C_VEL
LIN {X 0,Y 234.145,Z 631.323,A -85,B 0,C 180,E1 -20457,E2 -20457} C_VEL
LIN {X 0,Y 236.211,Z 620.177,A -85,B 0,C 180,E1 -20458.428,E2 -20458.428} C_VEL
LIN {X 0,Y 238.167,Z 607.522,A -85,B 0,C 180,E1 -20459.622,E2 -20459.622} C_VEL
LIN {X 0,Y 239.383,Z 595.876,A -85,B 0,C 180,E1 -20460.427,E2 -20460.427} C_VEL
LIN {X 0,Y 240.32,Z 583.641,A -85,B 0,C 180,E1 -20460.965,E2 -20460.965} C_VEL
LIN {X 0,Y 242.998,Z 516.06,A -85,B 0,C 180,E1 -20462.907,E2 -20462.907} C_VEL
LIN {X 0,Y 239.862,Z 496.141,A -85,B 0,C 180,E1 -20464.099,E2 -20464.099} C_VEL
LIN {X 0,Y 233.956,Z 482.666,A -85,B 0,C 180,E1 -20465.584,E2 -20465.584} C_VEL
LIN {X 0,Y 230.47,Z 475.32,A -85,B 0,C 180,E1 -20466.522,E2 -20466.522} C_VEL
LIN {X 0,Y 227.406,Z 464.434,A -85,B 0,C 180,E1 -20470.076,E2 -20470.076} C_VEL
LIN {X 0,Y 223.972,Z 454.426,A -85,B 0,C 180,E1 -20473.803,E2 -20473.803} C_VEL
LIN {X 0,Y 220.771,Z 445.974,A -85,B 0,C 180,E1 -20477.216,E2 -20477.216} C_VEL
LIN {X 0,Y 220.809,Z 445.983,A -85,B 0,C 180,E1 -20480.463,E2 -20480.463} C_VEL
LIN {X 0,Y 220.94,Z 446.089,A -85,B 0,C 180,E1 -20485,E2 -20485} C_VEL
LIN {X 0,Y 224.475,Z 463.021,A -85,B 0,C 180,E1 -20489.687,E2 -20489.687} C_VEL
LIN {X 0,Y 226.074,Z 470.827,A -85,B 0,C 180,E1 -20491.793,E2 -20491.793} C_VEL
LIN {X 0,Y 225.802,Z 476.414,A -85,B 0,C 180,E1 -20493.135,E2 -20493.135} C_VEL
LIN {X 0,Y 227.356,Z 497.248,A -85,B 0,C 180,E1 -20494.312,E2 -20494.312} C_VEL
LIN {X 0,Y 228.716,Z 510.536,A -85,B 0,C 180,E1 -20495.067,E2 -20495.067} C_VEL
LIN {X 0,Y 225.242,Z 587.453,A -85,B 0,C 180,E1 -20499.127,E2 -20499.127} C_VEL
LIN {X 0,Y 224.797,Z 594.299,A -85,B 0,C 180,E1 -20499.603,E2 -20499.603} C_VEL
LIN {X 0,Y 223.629,Z 599.826,A -85,B 0,C 180,E1 -20500.052,E2 -20500.052} C_VEL
LIN {X 0,Y 220.156,Z 608.539,A -85,B 0,C 180,E1 -20500.888,E2 -20500.888} C_VEL
LIN {X 0,Y 216.774,Z 617.07,A -85,B 0,C 180,E1 -20501.9,E2 -20501.9} C_VEL
LIN {X 0,Y 215.729,Z 622.239,A -85,B 0,C 180,E1 -20502.604,E2 -20502.604} C_VEL
LIN {X 0,Y 214.865,Z 633.234,A -85,B 0,C 180,E1 -20504.345,E2 -20504.345} C_VEL
LIN {X 0,Y 213.888,Z 644.013,A -85,B 0,C 180,E1 -20506.46,E2 -20506.46} C_VEL
LIN {X 0,Y 213.166,Z 652.989,A -85,B 0,C 180,E1 -20508.591,E2 -20508.591} C_VEL
LIN {X 0,Y 212.455,Z 662.756,A -85,B 0,C 180,E1 -20511.439,E2 -20511.439} C_VEL
LIN {X 0,Y 211.981,Z 670.667,A -85,B 0,C 180,E1 -20514.292,E2 -20514.292} C_VEL
LIN {X 0,Y 211.802,Z 677.002,A -85,B 0,C 180,E1 -20517.147,E2 -20517.147} C_VEL
LIN {X 0,Y 211.662,Z 681.974,A -85,B 0,C 180,E1 -20520,E2 -20520} C_VEL
LIN {X 0,Y 211.736,Z 685.799,A -85,B 0,C 180,E1 -20522.854,E2 -20522.854} C_VEL
LIN {X 0,Y 212.138,Z 689.146,A -85,B 0,C 180,E1 -20526.339,E2 -20526.339} C_VEL
LIN {X 0,Y 213.146,Z 690.975,A -85,B 0,C 180,E1 -20529.489,E2 -20529.489} C_VEL
LIN {X 0,Y 215.143,Z 691.715,A -85,B 0,C 180,E1 -20533.219,E2 -20533.219} C_VEL
LIN {X 0,Y 218.068,Z 690.963,A -85,B 0,C 180,E1 -20536.861,E2 -20536.861} C_VEL
LIN {X 0,Y 219.826,Z 690.009,A -85,B 0,C 180,E1 -20538.645,E2 -20538.645} C_VEL
LIN {X 0,Y 224.376,Z 686.877,A -85,B 0,C 180,E1 -20542.078,E2 -20542.078} C_VEL
LIN {X 0,Y 228.338,Z 683.466,A -85,B 0,C 180,E1 -20544.552,E2 -20544.552} C_VEL
LIN {X 0,Y 232.804,Z 679.054,A -85,B 0,C 180,E1 -20546.925,E2 -20546.925} C_VEL
LIN {X 0,Y 238.63,Z 672.545,A -85,B 0,C 180,E1 -20549.559,E2 -20549.559} C_VEL
LIN {X 0,Y 245.047,Z 664.333,A -85,B 0,C 180,E1 -20552.045,E2 -20552.045} C_VEL
LIN {X 0,Y 251.013,Z 655.634,A -85,B 0,C 180,E1 -20554.054,E2 -20554.054} C_VEL
LIN {X 0,Y 257.393,Z 645.186,A -85,B 0,C 180,E1 -20555.948,E2 -20555.948} C_VEL
LIN {X 0,Y 263.617,Z 633.289,A -85,B 0,C 180,E1 -20557.578,E2 -20557.578} C_VEL
LIN {X 0,Y 268.33,Z 622.94,A -85,B 0,C 180,E1 -20558.706,E2 -20558.706} C_VEL
LIN {X 0,Y 273.277,Z 609.905,A -85,B 0,C 180,E1 -20559.771,E2 -20559.771} C_VEL
LIN {X 0,Y 277.476,Z 596.373,A -85,B 0,C 180,E1 -20560.59,E2 -20560.59} C_VEL
LIN {X 0,Y 288.737,Z 549.812,A -85,B 0,C 180,E1 -20562.678,E2 -20562.678} C_VEL
LIN {X 0,Y 288.8,Z 549.337,A -85,B 0,C 180,E1 -20562.817,E2 -20562.817} C_VEL
LIN {X 0,Y 288.773,Z 547.706,A -85,B 0,C 180,E1 -20564.367,E2 -20564.367} C_VEL
LIN {X 0,Y 288.809,Z 547.429,A -85,B 0,C 180,E1 -20565.114,E2 -20565.114} C_VEL
LIN {X 0,Y 289.194,Z 547.453,A -85,B 0,C 180,E1 -20566.884,E2 -20566.884} C_VEL
LIN {X 0,Y 287.655,Z 553.918,A -85,B 0,C 180,E1 -20567.36,E2 -20567.36} C_VEL
LIN {X 0,Y 276.059,Z 601.495,A -85,B 0,C 180,E1 -20569.519,E2 -20569.519} C_VEL
LIN {X 0,Y 271.262,Z 616.315,A -85,B 0,C 180,E1 -20570.357,E2 -20570.357} C_VEL
LIN {X 0,Y 265.974,Z 629.33,A -85,B 0,C 180,E1 -20571.372,E2 -20571.372} C_VEL
LIN {X 0,Y 259.726,Z 642.384,A -85,B 0,C 180,E1 -20572.738,E2 -20572.738} C_VEL
LIN {X 0,Y 254.486,Z 651.945,A -85,B 0,C 180,E1 -20574.066,E2 -20574.066} C_VEL
LIN {X 0,Y 247.825,Z 662.689,A -85,B 0,C 180,E1 -20575.938,E2 -20575.938} C_VEL
LIN {X 0,Y 241.764,Z 671.467,A -85,B 0,C 180,E1 -20577.959,E2 -20577.959} C_VEL
LIN {X 0,Y 236.194,Z 678.793,A -85,B 0,C 180,E1 -20580.106,E2 -20580.106} C_VEL
LIN {X 0,Y 230.415,Z 685.685,A -85,B 0,C 180,E1 -20582.773,E2 -20582.773} C_VEL
LIN {X 0,Y 225.983,Z 690.45,A -85,B 0,C 180,E1 -20585.175,E2 -20585.175} C_VEL
LIN {X 0,Y 220.991,Z 695.266,A -85,B 0,C 180,E1 -20588.548,E2 -20588.548} C_VEL
LIN {X 0,Y 217.956,Z 697.805,A -85,B 0,C 180,E1 -20591.189,E2 -20591.189} C_VEL
LIN {X 0,Y 214.895,Z 699.815,A -85,B 0,C 180,E1 -20594.833,E2 -20594.833} C_VEL
LIN {X 0,Y 212.939,Z 700.353,A -85,B 0,C 180,E1 -20598.578,E2 -20598.578} C_VEL
LIN {X 0,Y 212.306,Z 700.046,A -85,B 0,C 180,E1 -20600.473,E2 -20600.473} C_VEL
LIN {X 0,Y 211.793,Z 698.976,A -85,B 0,C 180,E1 -20603.091,E2 -20603.091} C_VEL
LIN {X 0,Y 211.52,Z 700.839,A -85,B 0,C 180,E1 -20606.19,E2 -20606.19} C_VEL
LIN {X 0,Y 211.528,Z 701.455,A -85,B 0,C 180,E1 -20608.096,E2 -20608.096} C_VEL
LIN {X 0,Y 211.6,Z 701.673,A -85,B 0,C 180,E1 -20610,E2 -20610} C_VEL
LIN {X 0,Y 211.496,Z 701.443,A -85,B 0,C 180,E1 -20611.904,E2 -20611.904} C_VEL
LIN {X 0,Y 211.473,Z 700.552,A -85,B 0,C 180,E1 -20614.434,E2 -20614.434} C_VEL
LIN {X 0,Y 211.719,Z 698.362,A -85,B 0,C 180,E1 -20617.63,E2 -20617.63} C_VEL
LIN {X 0,Y 212.331,Z 695.378,A -85,B 0,C 180,E1 -20620.489,E2 -20620.489} C_VEL
LIN {X 0,Y 213.243,Z 691.328,A -85,B 0,C 180,E1 -20623.339,E2 -20623.339} C_VEL
LIN {X 0,Y 215.06,Z 685.097,A -85,B 0,C 180,E1 -20626.615,E2 -20626.615} C_VEL
LIN {X 0,Y 217.094,Z 678.303,A -85,B 0,C 180,E1 -20629.38,E2 -20629.38} C_VEL
LIN {X 0,Y 219.118,Z 671.2,A -85,B 0,C 180,E1 -20631.715,E2 -20631.715} C_VEL
LIN {X 0,Y 223.598,Z 666.025,A -85,B 0,C 180,E1 -20635.108,E2 -20635.108} C_VEL
LIN {X 0,Y 227.819,Z 660.993,A -85,B 0,C 180,E1 -20637.564,E2 -20637.564} C_VEL
LIN {X 0,Y 233.588,Z 653.832,A -85,B 0,C 180,E1 -20640.262,E2 -20640.262} C_VEL
LIN {X 0,Y 240.159,Z 645.006,A -85,B 0,C 180,E1 -20642.778,E2 -20642.778} C_VEL
LIN {X 0,Y 246.347,Z 635.943,A -85,B 0,C 180,E1 -20644.791,E2 -20644.791} C_VEL
LIN {X 0,Y 252.058,Z 626.993,A -85,B 0,C 180,E1 -20646.335,E2 -20646.335} C_VEL
LIN {X 0,Y 258.578,Z 615.591,A -85,B 0,C 180,E1 -20647.909,E2 -20647.909} C_VEL
LIN {X 0,Y 265.795,Z 601.166,A -85,B 0,C 180,E1 -20649.39,E2 -20649.39} C_VEL
LIN {X 0,Y 271.966,Z 586.51,A -85,B 0,C 180,E1 -20650.487,E2 -20650.487} C_VEL
LIN {X 0,Y 277.364,Z 570.475,A -85,B 0,C 180,E1 -20651.411,E2 -20651.411} C_VEL
LIN {X 0,Y 282.564,Z 549.5,A -85,B 0,C 180,E1 -20652.412,E2 -20652.412} C_VEL
LIN {X 0,Y 283.939,Z 542.483,A -85,B 0,C 180,E1 -20653.126,E2 -20653.126} C_VEL
LIN {X 0,Y 283.972,Z 540.608,A -85,B 0,C 180,E1 -20653.967,E2 -20653.967} C_VEL
LIN {X 0,Y 284.209,Z 537.83,A -85,B 0,C 180,E1 -20656.033,E2 -20656.033} C_VEL
LIN {X 0,Y 284.618,Z 536.987,A -85,B 0,C 180,E1 -20657.504,E2 -20657.504} C_VEL
LIN {X 0,Y 285.133,Z 536.839,A -85,B 0,C 180,E1 -20658.696,E2 -20658.696} C_VEL
LIN {X 0,Y 279.843,Z 558.553,A -85,B 0,C 180,E1 -20659.824,E2 -20659.824} C_VEL
LIN {X 0,Y 276.12,Z 570.809,A -85,B 0,C 180,E1 -20660.718,E2 -20660.718} C_VEL
LIN {X 0,Y 271.309,Z 583.477,A -85,B 0,C 180,E1 -20661.921,E2 -20661.921} C_VEL
LIN {X 0,Y 266.089,Z 594.921,A -85,B 0,C 180,E1 -20663.303,E2 -20663.303} C_VEL
LIN {X 0,Y 260.208,Z 605.784,A -85,B 0,C 180,E1 -20664.974,E2 -20664.974} C_VEL
LIN {X 0,Y 255.078,Z 614.053,A -85,B 0,C 180,E1 -20666.561,E2 -20666.561} C_VEL
LIN {X 0,Y 249.24,Z 622.301,A -85,B 0,C 180,E1 -20668.556,E2 -20668.556} C_VEL
LIN {X 0,Y 243.846,Z 629.036,A -85,B 0,C 180,E1 -20670.662,E2 -20670.662} C_VEL
LIN {X 0,Y 238.772,Z 634.569,A -85,B 0,C 180,E1 -20672.856,E2 -20672.856} C_VEL
LIN {X 0,Y 234.14,Z 638.975,A -85,B 0,C 180,E1 -20675.151,E2 -20675.151} C_VEL
LIN {X 0,Y 231.264,Z 641.368,A -85,B 0,C 180,E1 -20676.73,E2 -20676.73} C_VEL
LIN {X 0,Y 228.541,Z 643.338,A -85,B 0,C 180,E1 -20678.345,E2 -20678.345} C_VEL
LIN {X 0,Y 223.658,Z 646.034,A -85,B 0,C 180,E1 -20681.686,E2 -20681.686} C_VEL
LIN {X 0,Y 221.547,Z 646.796,A -85,B 0,C 180,E1 -20683.411,E2 -20683.411} C_VEL
LIN {X 0,Y 219.643,Z 647.146,A -85,B 0,C 180,E1 -20685.168,E2 -20685.168} C_VEL
LIN {X 0,Y 216.61,Z 646.645,A -85,B 0,C 180,E1 -20688.774,E2 -20688.774} C_VEL
LIN {X 0,Y 214.464,Z 644.617,A -85,B 0,C 180,E1 -20692.468,E2 -20692.468} C_VEL
LIN {X 0,Y 213.261,Z 642.032,A -85,B 0,C 180,E1 -20695.274,E2 -20695.274} C_VEL
LIN {X 0,Y 212.499,Z 638.472,A -85,B 0,C 180,E1 -20698.105,E2 -20698.105} C_VEL
LIN {X 0,Y 212.243,Z 633.894,A -85,B 0,C 180,E1 -20700.949,E2 -20700.949} C_VEL
LIN {X 0,Y 212.465,Z 627.121,A -85,B 0,C 180,E1 -20704.268,E2 -20704.268} C_VEL
LIN {X 0,Y 212.666,Z 620.245,A -85,B 0,C 180,E1 -20706.948,E2 -20706.948} C_VEL
LIN {X 0,Y 213.146,Z 612.38,A -85,B 0,C 180,E1 -20709.489,E2 -20709.489} C_VEL
LIN {X 0,Y 213.823,Z 603.615,A -85,B 0,C 180,E1 -20711.855,E2 -20711.855} C_VEL
LIN {X 0,Y 214.687,Z 593.04,A -85,B 0,C 180,E1 -20714.213,E2 -20714.213} C_VEL
LIN {X 0,Y 215.704,Z 581.449,A -85,B 0,C 180,E1 -20716.321,E2 -20716.321} C_VEL
LIN {X 0,Y 216.575,Z 570.436,A -85,B 0,C 180,E1 -20717.956,E2 -20717.956} C_VEL
LIN {X 0,Y 217.486,Z 556.255,A -85,B 0,C 180,E1 -20719.589,E2 -20719.589} C_VEL
LIN {X 0,Y 218.264,Z 541.964,A -85,B 0,C 180,E1 -20720.805,E2 -20720.805} C_VEL
LIN {X 0,Y 219.206,Z 516.476,A -85,B 0,C 180,E1 -20722.286,E2 -20722.286} C_VEL
LIN {X 0,Y 221.128,Z 472.758,A -85,B 0,C 180,E1 -20724.678,E2 -20724.678} C_VEL
LIN {X 0,Y 213.935,Z 447.289,A -85,B 0,C 180,E1 -20726.414,E2 -20726.414} C_VEL
LIN {X 0,Y 213.863,Z 446.841,A -85,B 0,C 180,E1 -20726.499,E2 -20726.499} C_VEL
LIN {X 0,Y 213.769,Z 446.834,A -85,B 0,C 180,E1 -20731.738,E2 -20731.738} C_VEL
LIN {X 0,Y 213.746,Z 446.85,A -85,B 0,C 180,E1 -20736.288,E2 -20736.288} C_VEL
LIN {X 0,Y 213.728,Z 446.841,A -85,B 0,C 180,E1 -20741.278,E2 -20741.278} C_VEL
LIN {X 0,Y 217.329,Z 456.37,A -85,B 0,C 180,E1 -20745.352,E2 -20745.352} C_VEL
LIN {X 0,Y 220.266,Z 464.702,A -85,B 0,C 180,E1 -20748.573,E2 -20748.573} C_VEL
LIN {X 0,Y 223.154,Z 474.326,A -85,B 0,C 180,E1 -20751.939,E2 -20751.939} C_VEL
LIN {X 0,Y 223.616,Z 475.906,A -85,B 0,C 180,E1 -20752.379,E2 -20752.379} C_VEL
LIN {X 0,Y 229.847,Z 488.749,A -85,B 0,C 180,E1 -20754.059,E2 -20754.059} C_VEL
LIN {X 0,Y 234.265,Z 499.136,A -85,B 0,C 180,E1 -20755.224,E2 -20755.224} C_VEL
LIN {X 0,Y 236.994,Z 517.847,A -85,B 0,C 180,E1 -20756.355,E2 -20756.355} C_VEL
LIN {X 0,Y 234.049,Z 586.053,A -85,B 0,C 180,E1 -20758.362,E2 -20758.362} C_VEL
LIN {X 0,Y 232.914,Z 599.172,A -85,B 0,C 180,E1 -20759.013,E2 -20759.013} C_VEL
LIN {X 0,Y 231.415,Z 611.107,A -85,B 0,C 180,E1 -20759.927,E2 -20759.927} C_VEL
LIN {X 0,Y 229.454,Z 622.81,A -85,B 0,C 180,E1 -20761.157,E2 -20761.157} C_VEL
LIN {X 0,Y 227.021,Z 634.848,A -85,B 0,C 180,E1 -20762.83,E2 -20762.83} C_VEL
LIN {X 0,Y 224.441,Z 645.438,A -85,B 0,C 180,E1 -20764.745,E2 -20764.745} C_VEL
LIN {X 0,Y 222.198,Z 654.1,A -85,B 0,C 180,E1 -20766.714,E2 -20766.714} C_VEL
LIN {X 0,Y 219.529,Z 663.494,A -85,B 0,C 180,E1 -20769.381,E2 -20769.381} C_VEL
LIN {X 0,Y 217.121,Z 670.96,A -85,B 0,C 180,E1 -20772.091,E2 -20772.091} C_VEL
LIN {X 0,Y 215.275,Z 676.944,A -85,B 0,C 180,E1 -20774.86,E2 -20774.86} C_VEL
LIN {X 0,Y 213.76,Z 681.676,A -85,B 0,C 180,E1 -20777.66,E2 -20777.66} C_VEL
LIN {X 0,Y 212.72,Z 685.291,A -85,B 0,C 180,E1 -20780.491,E2 -20780.491} C_VEL
LIN {X 0,Y 212.239,Z 687.151,A -85,B 0,C 180,E1 -20782.389,E2 -20782.389} C_VEL
LIN {X 0,Y 211.893,Z 688.568,A -85,B 0,C 180,E1 -20784.289,E2 -20784.289} C_VEL
LIN {X 0,Y 211.567,Z 690.171,A -85,B 0,C 180,E1 -20788.096,E2 -20788.096} C_VEL
LIN {X 0,Y 211.554,Z 690.402,A -85,B 0,C 180,E1 -20790,E2 -20790} C_VEL
LIN {X 0,Y 211.566,Z 690.205,A -85,B 0,C 180,E1 -20791.904,E2 -20791.904} C_VEL
LIN {X 0,Y 211.893,Z 688.646,A -85,B 0,C 180,E1 -20795.711,E2 -20795.711} C_VEL
LIN {X 0,Y 212.235,Z 687.273,A -85,B 0,C 180,E1 -20797.612,E2 -20797.612} C_VEL
LIN {X 0,Y 212.998,Z 684.392,A -85,B 0,C 180,E1 -20800.456,E2 -20800.456} C_VEL
LIN {X 0,Y 214.17,Z 680.472,A -85,B 0,C 180,E1 -20803.28,E2 -20803.28} C_VEL
LIN {X 0,Y 215.807,Z 675.387,A -85,B 0,C 180,E1 -20806.07,E2 -20806.07} C_VEL
LIN {X 0,Y 217.846,Z 668.977,A -85,B 0,C 180,E1 -20808.821,E2 -20808.821} C_VEL
LIN {X 0,Y 220.372,Z 661.005,A -85,B 0,C 180,E1 -20811.516,E2 -20811.516} C_VEL
LIN {X 0,Y 222.616,Z 652.918,A -85,B 0,C 180,E1 -20813.718,E2 -20813.718} C_VEL
LIN {X 0,Y 224.889,Z 643.941,A -85,B 0,C 180,E1 -20815.697,E2 -20815.697} C_VEL
LIN {X 0,Y 227.548,Z 632.875,A -85,B 0,C 180,E1 -20817.6,E2 -20817.6} C_VEL
LIN {X 0,Y 229.676,Z 622.078,A -85,B 0,C 180,E1 -20819.063,E2 -20819.063} C_VEL
LIN {X 0,Y 231.729,Z 610.133,A -85,B 0,C 180,E1 -20820.279,E2 -20820.279} C_VEL
LIN {X 0,Y 233.191,Z 596.856,A -85,B 0,C 180,E1 -20821.262,E2 -20821.262} C_VEL
LIN {X 0,Y 234.28,Z 583.722,A -85,B 0,C 180,E1 -20821.856,E2 -20821.856} C_VEL
LIN {X 0,Y 237.059,Z 517.129,A -85,B 0,C 180,E1 -20823.804,E2 -20823.804} C_VEL
LIN {X 0,Y 234.272,Z 499.037,A -85,B 0,C 180,E1 -20824.925,E2 -20824.925} C_VEL
LIN {X 0,Y 228.671,Z 486.073,A -85,B 0,C 180,E1 -20826.408,E2 -20826.408} C_VEL
LIN {X 0,Y 223.442,Z 475.32,A -85,B 0,C 180,E1 -20827.898,E2 -20827.898} C_VEL
LIN {X 0,Y 220.872,Z 466.59,A -85,B 0,C 180,E1 -20830.913,E2 -20830.913} C_VEL
LIN {X 0,Y 218.217,Z 458.583,A -85,B 0,C 180,E1 -20833.939,E2 -20833.939} C_VEL
LIN {X 0,Y 214.551,Z 449.395,A -85,B 0,C 180,E1 -20837.816,E2 -20837.816} C_VEL
LIN {X 0,Y 213.735,Z 446.848,A -85,B 0,C 180,E1 -20839.011,E2 -20839.011} C_VEL
LIN {X 0,Y 213.844,Z 446.867,A -85,B 0,C 180,E1 -20844.667,E2 -20844.667} C_VEL
LIN {X 0,Y 216.86,Z 461.312,A -85,B 0,C 180,E1 -20848.766,E2 -20848.766} C_VEL
LIN {X 0,Y 219.097,Z 472.177,A -85,B 0,C 180,E1 -20851.762,E2 -20851.762} C_VEL
LIN {X 0,Y 218.794,Z 476.58,A -85,B 0,C 180,E1 -20852.824,E2 -20852.824} C_VEL
LIN {X 0,Y 220.342,Z 497.853,A -85,B 0,C 180,E1 -20854.072,E2 -20854.072} C_VEL
LIN {X 0,Y 221.671,Z 511.008,A -85,B 0,C 180,E1 -20854.846,E2 -20854.846} C_VEL
LIN {X 0,Y 218.102,Z 588.007,A -85,B 0,C 180,E1 -20859.105,E2 -20859.105} C_VEL
LIN {X 0,Y 217.355,Z 601.353,A -85,B 0,C 180,E1 -20860.168,E2 -20860.168} C_VEL
LIN {X 0,Y 216.393,Z 614.186,A -85,B 0,C 180,E1 -20861.539,E2 -20861.539} C_VEL
LIN {X 0,Y 215.729,Z 622.239,A -85,B 0,C 180,E1 -20862.604,E2 -20862.604} C_VEL
LIN {X 0,Y 214.633,Z 627.312,A -85,B 0,C 180,E1 -20863.356,E2 -20863.356} C_VEL
LIN {X 0,Y 211.165,Z 635.081,A -85,B 0,C 180,E1 -20864.728,E2 -20864.728} C_VEL
LIN {X 0,Y 207.668,Z 642.44,A -85,B 0,C 180,E1 -20866.301,E2 -20866.301} C_VEL
LIN {X 0,Y 206.541,Z 646.882,A -85,B 0,C 180,E1 -20867.351,E2 -20867.351} C_VEL
LIN {X 0,Y 205.71,Z 657.539,A -85,B 0,C 180,E1 -20870.164,E2 -20870.164} C_VEL
LIN {X 0,Y 205.104,Z 666.736,A -85,B 0,C 180,E1 -20873.211,E2 -20873.211} C_VEL
LIN {X 0,Y 204.79,Z 673.634,A -85,B 0,C 180,E1 -20876.064,E2 -20876.064} C_VEL
LIN {X 0,Y 204.672,Z 679.34,A -85,B 0,C 180,E1 -20879.016,E2 -20879.016} C_VEL
LIN {X 0,Y 204.669,Z 683.832,A -85,B 0,C 180,E1 -20881.968,E2 -20881.968} C_VEL
LIN {X 0,Y 204.752,Z 686.226,A -85,B 0,C 180,E1 -20883.936,E2 -20883.936} C_VEL
LIN {X 0,Y 205.069,Z 688.544,A -85,B 0,C 180,E1 -20886.345,E2 -20886.345} C_VEL
LIN {X 0,Y 206.138,Z 690.826,A -85,B 0,C 180,E1 -20889.815,E2 -20889.815} C_VEL
LIN {X 0,Y 208.237,Z 691.974,A -85,B 0,C 180,E1 -20893.665,E2 -20893.665} C_VEL
LIN {X 0,Y 211.313,Z 691.575,A -85,B 0,C 180,E1 -20897.417,E2 -20897.417} C_VEL
LIN {X 0,Y 213.156,Z 690.821,A -85,B 0,C 180,E1 -20899.251,E2 -20899.251} C_VEL
LIN {X 0,Y 217.928,Z 688.169,A -85,B 0,C 180,E1 -20902.767,E2 -20902.767} C_VEL
LIN {X 0,Y 223.56,Z 683.882,A -85,B 0,C 180,E1 -20906.111,E2 -20906.111} C_VEL
LIN {X 0,Y 228.389,Z 679.529,A -85,B 0,C 180,E1 -20908.488,E2 -20908.488} C_VEL
LIN {X 0,Y 234.637,Z 673.159,A -85,B 0,C 180,E1 -20911.11,E2 -20911.11} C_VEL
LIN {X 0,Y 241.485,Z 665.039,A -85,B 0,C 180,E1 -20913.571,E2 -20913.571} C_VEL
LIN {X 0,Y 247.817,Z 656.598,A -85,B 0,C 180,E1 -20915.547,E2 -20915.547} C_VEL
LIN {X 0,Y 254.527,Z 646.312,A -85,B 0,C 180,E1 -20917.407,E2 -20917.407} C_VEL
LIN {X 0,Y 260.473,Z 635.917,A -85,B 0,C 180,E1 -20918.853,E2 -20918.853} C_VEL
LIN {X 0,Y 266.004,Z 624.655,A -85,B 0,C 180,E1 -20920.092,E2 -20920.092} C_VEL
LIN {X 0,Y 271.175,Z 612.23,A -85,B 0,C 180,E1 -20921.12,E2 -20921.12} C_VEL
LIN {X 0,Y 275.048,Z 600.796,A -85,B 0,C 180,E1 -20921.834,E2 -20921.834} C_VEL
LIN {X 0,Y 280.304,Z 581.13,A -85,B 0,C 180,E1 -20922.763,E2 -20922.763} C_VEL
LIN {X 0,Y 286.861,Z 555.073,A -85,B 0,C 180,E1 -20923.887,E2 -20923.887} C_VEL
LIN {X 0,Y 286.988,Z 554.277,A -85,B 0,C 180,E1 -20925.249,E2 -20925.249} C_VEL
LIN {X 0,Y 287.055,Z 554.35,A -85,B 0,C 180,E1 -20925.943,E2 -20925.943} C_VEL
LIN {X 0,Y 274.752,Z 602.041,A -85,B 0,C 180,E1 -20928.067,E2 -20928.067} C_VEL
LIN {X 0,Y 269.892,Z 616.093,A -85,B 0,C 180,E1 -20928.84,E2 -20928.84} C_VEL
LIN {X 0,Y 264.249,Z 629.253,A -85,B 0,C 180,E1 -20929.837,E2 -20929.837} C_VEL
LIN {X 0,Y 258.315,Z 640.998,A -85,B 0,C 180,E1 -20931.011,E2 -20931.011} C_VEL
LIN {X 0,Y 252.713,Z 650.647,A -85,B 0,C 180,E1 -20932.278,E2 -20932.278} C_VEL
